// TIA Portal V15.1 export
// export: Created 2024-06-21T08:41:18.4574787Z, ExportSetting WithDefaults, DisplayName Totally Integrated Automation Portal, DisplayVersion V15.1 Update 5, DisplayName TIA Portal Openness, DisplayVersion V15.1 Update 5, DisplayName SINAMICS Startdrive Advanced, DisplayVersion V15.1, DisplayName G130, G150, S120, S150, SINAMICS MV, S210, DisplayVersion V15.1, DisplayName G110M, G120, G120C, G120D, G120P, DisplayVersion V15.1, DisplayName STEP 7 Professional, DisplayVersion V15.1 Update 5, DisplayName STEP 7 Safety, DisplayVersion V15.1, DisplayName WinCC Professional, DisplayVersion V15.1 Update 5, DisplayName SIMATIC Visualization Architect, DisplayVersion V15.1
FUNCTION_BLOCK "LGBLiftTable2Pos1S3Det-C"   // FB6675, FBD
TITLE = LMovUnit2Pos2Det2W2S-G120CU240PN / LMovUnit2Pos2W2S-G120CU240PN / LGBLiftTable2Pos1S3Det-C
{ S7_Optimized_Access := 'TRUE' }
AUTHOR : VCC
FAMILY : Tooling
VERSION : 0.0.0.0
// =============================================================================
// This module will be used for a unit with 2 stop positions, 2 speeds and controlled by a
// Siemens G120 PN frequency converter.
// It will get commands from higher level, evaluate the status of the interlock
// and give a finished in return when the task is completed.
// It will get commands from higher level, evaluate the status of the interlock
// and give a finished in return when the task is completed.
// ============================================================================
// stored: AutoNumber false, IsIECCheckEnabled false, IsRetainMemResEnabled false, MemoryReserve 100, SetENOAutomatically False, UDAEnableTagReadback false
   VAR_INPUT
      I_PosSet { ExternalAccessible := 'False'; ExternalVisible := 'False'; ExternalWritable := 'False'} : Bool;   // Position Set detection or summary / Position Set Detection / Position Set Detection 1
      I_PosSetCheck { ExternalAccessible := 'False'; ExternalVisible := 'False'; ExternalWritable := 'False'} : Bool;   // Low Speed Set / Low Speed Detection Set / Position Set Detection 2
      I_PosRes { ExternalAccessible := 'False'; ExternalVisible := 'False'; ExternalWritable := 'False'} : Bool;   // Position Reset detection or summary / Position Reset Detection / Position Reset Detection 1
      I_PosResCheck { ExternalAccessible := 'False'; ExternalVisible := 'False'; ExternalWritable := 'False'} : Bool;   // Low Speed Res / Low Speed Detection Reset / Position Reset Detection 2
      I_BrakeReleased { ExternalAccessible := 'False'; ExternalVisible := 'False'; ExternalWritable := 'False'} : Bool;   // Feedback from brake contactor
      I_SetBegin { ExternalAccessible := 'False'; ExternalVisible := 'False'; ExternalWritable := 'False'} : Bool;   // Function Set begin selection
      I_ResBegin { ExternalAccessible := 'False'; ExternalVisible := 'False'; ExternalWritable := 'False'} : Bool;   // Function Reset begin selection
      I_PBSet { ExternalAccessible := 'False'; ExternalVisible := 'False'; ExternalWritable := 'False'} : Bool;   // Push button for Set direction (used in manual with button OP panels ) / Push button for Set direction used in manual
      I_PBReset { ExternalAccessible := 'False'; ExternalVisible := 'False'; ExternalWritable := 'False'} : Bool;   // Push button for reset direcion (used in manual with pushbutton OP panels) / Push button for reset direcion used in manual
      I_SetIntlkOK { ExternalAccessible := 'False'; ExternalVisible := 'False'; ExternalWritable := 'False'} : Bool;   // Set Interlock
      I_ResIntlkOK { ExternalAccessible := 'False'; ExternalVisible := 'False'; ExternalWritable := 'False'} : Bool;   // Reset Interlock
      I_MotorProtection { ExternalAccessible := 'False'; ExternalVisible := 'False'; ExternalWritable := 'False'} : Bool;   // Motor protection
      I_SafetySwitch { ExternalAccessible := 'False'; ExternalVisible := 'False'; ExternalWritable := 'False'} : Bool;   // Safety switch
      I_SafetyOk { ExternalAccessible := 'False'; ExternalVisible := 'False'; ExternalWritable := 'False'} : Bool;   // Safety Ok
      I_MotionStopOk { ExternalAccessible := 'False'; ExternalVisible := 'False'; ExternalWritable := 'False'} : Bool;   // Safety Ok / The motion stop is Ok
   END_VAR
   VAR_OUTPUT
      O_SetContactor { ExternalAccessible := 'False'; ExternalVisible := 'False'; ExternalWritable := 'False'} : Bool;   // Activate set contactor
      O_ResetContactor { ExternalAccessible := 'False'; ExternalVisible := 'False'; ExternalWritable := 'False'} : Bool;   // Activate Reset contactor
      O_ReleaseBrakeContactor { ExternalAccessible := 'False'; ExternalVisible := 'False'; ExternalWritable := 'False'} : Bool;   // Release Brake
      O_Active { ExternalAccessible := 'False'; ExternalVisible := 'False'; ExternalWritable := 'False'} : Bool;   // Motor Loop Active / Motor Active
      O_SetPos { ExternalAccessible := 'False'; ExternalVisible := 'False'; ExternalWritable := 'False'} : Bool;   // Summary In Position Set / In Position Set
      O_ResPos { ExternalAccessible := 'False'; ExternalVisible := 'False'; ExternalWritable := 'False'} : Bool;   // Summary In Position Reset / In Position Reset
      O_FuncRunning { ExternalAccessible := 'False'; ExternalVisible := 'False'; ExternalWritable := 'False'} : Bool;   // Signal that the function is busy
      O_SetFinished { ExternalAccessible := 'False'; ExternalVisible := 'False'; ExternalWritable := 'False'} : Bool;   // Function Set finished to Master Sequencing
      O_ResFinished { ExternalAccessible := 'False'; ExternalVisible := 'False'; ExternalWritable := 'False'} : Bool;   // Function Reset finished to Master Sequencing
      O_LEDSet { ExternalAccessible := 'False'; ExternalVisible := 'False'; ExternalWritable := 'False'} : Bool;   // Ledindication / Led indication for Set
      O_LEDRes { ExternalAccessible := 'False'; ExternalVisible := 'False'; ExternalWritable := 'False'} : Bool;   // Ledindication / Led indication for Reset
      O_AlarmABCondition { ExternalAccessible := 'False'; ExternalVisible := 'False'; ExternalWritable := 'False'} : Bool;   // Alarm AB condition
      O_AlarmA { ExternalAccessible := 'False'; ExternalVisible := 'False'; ExternalWritable := 'False'} : Bool;   // Summation Alarm A of roller. / Alarm A
      O_AlarmB { ExternalAccessible := 'False'; ExternalVisible := 'False'; ExternalWritable := 'False'} : Bool;   // Summation Alarm B of roller. / Alarm B
      O_AlarmC { ExternalAccessible := 'False'; ExternalVisible := 'False'; ExternalWritable := 'False'} : Bool;   // Summation Alarm C of roller. / Alarm C
      O_AlarmD { ExternalAccessible := 'False'; ExternalVisible := 'False'; ExternalWritable := 'False'} : Bool;   // Summation Alarm D of roller. / Alarm D
      H_AlarmDWord { ExternalAccessible := 'False'; ExternalVisible := 'False'; ExternalWritable := 'False'} : DWord;   // HMI Animation of the alarms of the roller / Alarm Word
   END_VAR
   VAR_IN_OUT
      IO_Modes : "Modes";   // Modes
      C_Config : "LiftTable2Pos1S3Det-C-Config";   // Config
      H_HMI : "H_HMI";   // Animation
      "H_GBLiftTable2Pos1S3Det-C" : "H_GBLiftTable2Pos1S3Det-C";   // Animation
   END_VAR
   VAR
      _MovFunc2Pos { ExternalAccessible := 'False'; ExternalVisible := 'False'; ExternalWritable := 'False'} : "LMovFnc2Pos";   // Move function 2 positioner / FB
      _StopPos { ExternalAccessible := 'False'; ExternalVisible := 'False'; ExternalWritable := 'False'} : "L2StopPos";   // FB
      _Motor { ExternalAccessible := 'False'; ExternalVisible := 'False'; ExternalWritable := 'False'} : "LGBMotor2W1S-C";   // FB
      _SetDetMissing { ExternalAccessible := 'False'; ExternalVisible := 'False'; ExternalWritable := 'False'} : "LTimer";   // Timer
      _ResDetMissing { ExternalAccessible := 'False'; ExternalVisible := 'False'; ExternalWritable := 'False'} : "LTimer";   // Timer
      H_FncSelInHMI { ExternalAccessible := 'False'; ExternalVisible := 'False'; ExternalWritable := 'False'} : Bool;
      AA_MotorProtection { ExternalAccessible := 'False'; ExternalVisible := 'False'; ExternalWritable := 'False'} : Bool;   // Motor protection alarm / Motorprotection Not Ok / Motor Protection Tripped / Motorskyddsbrytare Ej Ok
      AA_SafetySwitch { ExternalAccessible := 'False'; ExternalVisible := 'False'; ExternalWritable := 'False'} : Bool;   // Safety Switch alarm / Safety Switch Not Ok / Säkerhetsbrytare Ej Ok
      AB_BrakeFbk { ExternalAccessible := 'False'; ExternalVisible := 'False'; ExternalWritable := 'False'} : Bool;   // Safety Switch Not Ok / Brake feedback Nok / Säkerhetsbrytare Ej Ok
      AB_KeepPosSetAlm { ExternalAccessible := 'False'; ExternalVisible := 'False'; ExternalWritable := 'False'} : Bool;   // 0000: Keep position set alarm / Position Supervision Set Position / Lost Set Position / Positionsövervakning Set Läge
      AB_KeepPosResAlm { ExternalAccessible := 'False'; ExternalVisible := 'False'; ExternalWritable := 'False'} : Bool;   // 0000: Keep position reset alarm / Position Supervision Reset Position / Lost Reset Position / Positionsövervakning Reset Läge
      AB_OvtSetAlm { ExternalAccessible := 'False'; ExternalVisible := 'False'; ExternalWritable := 'False'} : Bool;   // 0000: Overtime set alarm / Timeout Set / TimeOut Set Direction / Tidsövervakning Set
      AB_OvtResAlm { ExternalAccessible := 'False'; ExternalVisible := 'False'; ExternalWritable := 'False'} : Bool;   // 0000: Overtime reset alarm / Timeout Reset / TimeOut Reset Direction / Tidsövervakning Reset
      AB_TwoDetAlm { ExternalAccessible := 'False'; ExternalVisible := 'False'; ExternalWritable := 'False'} : Bool;   // 0000: Two detection alarm / Set Reset Activated Simultaneously / Detection Set & Reset Activated Simultaneously / Set Reset Påverkade Samtidigt
      AB_SetDet1Missing { ExternalAccessible := 'False'; ExternalVisible := 'False'; ExternalWritable := 'False'} : Bool;   // 0000: Two detection alarm / Set Detector 1 Signal Missing / Set Detector Signal Missing / Setgivare 1 signal saknas
      AB_SetDet2Missing { ExternalAccessible := 'False'; ExternalVisible := 'False'; ExternalWritable := 'False'} : Bool;   // 0000: Two detection alarm / Set Detector 2 Signal Missing / Set Check Detector Signal Missing / Setgivare 2 signal saknas
      AB_ResDet1Missing { ExternalAccessible := 'False'; ExternalVisible := 'False'; ExternalWritable := 'False'} : Bool;   // 0000: Two detection alarm / Resetgivare 1 signal saknas / Reset Detector Signal Missing
      AB_ResDet2Missing { ExternalAccessible := 'False'; ExternalVisible := 'False'; ExternalWritable := 'False'} : Bool;   // 0000: Two detection alarm / Resetgivare 2 signal saknas / Reset Check Detector Signal Missing
      AC_KeepPosSetAlm { ExternalAccessible := 'False'; ExternalVisible := 'False'; ExternalWritable := 'False'} : Bool;   // 0000: Keep position set alarm / Lost Set Position / Tappat Set Position
      AC_KeepPosResAlm { ExternalAccessible := 'False'; ExternalVisible := 'False'; ExternalWritable := 'False'} : Bool;   // 0000: Keep position reset alarm / Lost Reset Position / Tappat Reset Position
      AC_OvtSetAlm { ExternalAccessible := 'False'; ExternalVisible := 'False'; ExternalWritable := 'False'} : Bool;   // 0000: Overtime set alarm / Timeout Set / TimeOut Set Direction / Tidsövervakning Set
      AC_OvtResAlm { ExternalAccessible := 'False'; ExternalVisible := 'False'; ExternalWritable := 'False'} : Bool;   // 0000: Overtime reset alarm / Timeout Reset / TimeOut Reset Direction / Tidsövervakning Reset
      AC_TwoDetAlm { ExternalAccessible := 'False'; ExternalVisible := 'False'; ExternalWritable := 'False'} : Bool;   // 0000: Two detection alarm / Set Reset Activated Simultaneously / Detection Set & Reset Activated Simultaneously / Set Reset Påverkade Samtidigt
      AC_SetDet1Missing { ExternalAccessible := 'False'; ExternalVisible := 'False'; ExternalWritable := 'False'} : Bool;   // 0000: Two detection alarm / Set Detector 1 Signal Missing / Set Detector Signal Missing / Setgivare 1 signal saknas
      AC_SetDet2Missing { ExternalAccessible := 'False'; ExternalVisible := 'False'; ExternalWritable := 'False'} : Bool;   // 0000: Two detection alarm / Set Detector 2 Signal Missing / Set Check Detector Signal Missing / Setgivare 2 signal saknas
      AC_ResDet1Missing { ExternalAccessible := 'False'; ExternalVisible := 'False'; ExternalWritable := 'False'} : Bool;   // 0000: Two detection alarm / Resetgivare 1 signal saknas / Reset Detector Signal Missing
      AC_ResDet2Missing { ExternalAccessible := 'False'; ExternalVisible := 'False'; ExternalWritable := 'False'} : Bool;   // 0000: Two detection alarm / Resetgivare 2 signal saknas / Reset Check Detector Signal Missing
      AD_OvtSetWarn { ExternalAccessible := 'False'; ExternalVisible := 'False'; ExternalWritable := 'False'} : Bool;   // 0000: Overtime set warning / Timeout Set / TimeOut Set Direction / Tidsövervakning Set
      AD_OvtResWarn { ExternalAccessible := 'False'; ExternalVisible := 'False'; ExternalWritable := 'False'} : Bool;   // 0000: Overtime reset warning / Timeout Reset / TimeOut Reset Direction / Tidsövervakning Reset
      AD_IntlkSetAlm { ExternalAccessible := 'False'; ExternalVisible := 'False'; ExternalWritable := 'False'} : Bool;   // 0000: Interlock Set alarm / Interlock Set
      AD_IntlkResAlm { ExternalAccessible := 'False'; ExternalVisible := 'False'; ExternalWritable := 'False'} : Bool;   // 0000: Interlock Reset alarm / Interlock Reset
      AD_MotionStop { ExternalAccessible := 'False'; ExternalVisible := 'False'; ExternalWritable := 'False'} : Bool;   // Motion Stop
      AC_ConfigCalibrationAlm { ExternalAccessible := 'False'; ExternalVisible := 'False'; ExternalWritable := 'False'} : Bool;   // The Config values for Warming/Alarm time must be ALL zero or ALL different from zero
      AD_CalibrationWarn { ExternalAccessible := 'False'; ExternalVisible := 'False'; ExternalWritable := 'False'} : Bool;   // No High speed selected so Calibration is not possible
      SafetyOk { ExternalAccessible := 'False'; ExternalVisible := 'False'; ExternalWritable := 'False'} : Bool;   // Safety Ok
      SetPos { ExternalAccessible := 'False'; ExternalVisible := 'False'; ExternalWritable := 'False'} : Bool;   // Set position
      ResPos { ExternalAccessible := 'False'; ExternalVisible := 'False'; ExternalWritable := 'False'} : Bool;   // Reset position
      AlarmA { ExternalAccessible := 'False'; ExternalVisible := 'False'; ExternalWritable := 'False'} : Bool;   // Summation Alarm A / Alarm A
      AlarmB { ExternalAccessible := 'False'; ExternalVisible := 'False'; ExternalWritable := 'False'} : Bool;   // Summation Alarm B / Alarm B
      AlarmC { ExternalAccessible := 'False'; ExternalVisible := 'False'; ExternalWritable := 'False'} : Bool;   // Summation Alarm C / Alarm C
      AlarmD { ExternalAccessible := 'False'; ExternalVisible := 'False'; ExternalWritable := 'False'} : Bool;   // Summation Alarm D / Alarm D
      SetIntlkOK { ExternalAccessible := 'False'; ExternalVisible := 'False'; ExternalWritable := 'False'} : Bool;   // Set Interlock
      ResIntlkOK { ExternalAccessible := 'False'; ExternalVisible := 'False'; ExternalWritable := 'False'} : Bool;   // Reset Interlock
      FuncRunning { ExternalAccessible := 'False'; ExternalVisible := 'False'; ExternalWritable := 'False'} : Bool;   // Function running
      MovFuncAlmCond { ExternalAccessible := 'False'; ExternalVisible := 'False'; ExternalWritable := 'False'} : Bool;   // Move function alarm condition / Move function Alarm Condition
      StopPosAlmCond { ExternalAccessible := 'False'; ExternalVisible := 'False'; ExternalWritable := 'False'} : Bool;   // Stop posistion alarm condition / Stop posistion Alarm Condition
      KeepPosSetAlm { ExternalAccessible := 'False'; ExternalVisible := 'False'; ExternalWritable := 'False'} : Bool;   // Keep position set alarm / Alarm Keep Position Set Position / Larm Positions Övervakning Set Läge
      KeepPosResAlm { ExternalAccessible := 'False'; ExternalVisible := 'False'; ExternalWritable := 'False'} : Bool;   // Keep position reset alarm / Position Supervision Reset Position / Positions Övervakning Reset Läge
      OvtSetAlm { ExternalAccessible := 'False'; ExternalVisible := 'False'; ExternalWritable := 'False'} : Bool;   // Overtime set alarm / Timeout Set / Tidsövervakning Set
      OvtResAlm { ExternalAccessible := 'False'; ExternalVisible := 'False'; ExternalWritable := 'False'} : Bool;   // Overtime reset alarm / Overtime reset Alarm
      TwoDetAlm { ExternalAccessible := 'False'; ExternalVisible := 'False'; ExternalWritable := 'False'} : Bool;   // Two detection alarm / Set Reset Activated Simultaneously / Set Reset Påverkade Samtidigt
      OneSetDetMissing { ExternalAccessible := 'False'; ExternalVisible := 'False'; ExternalWritable := 'False'} : Bool;   // Two detection alarm / One Set detector is missing
      OneResDetMissing { ExternalAccessible := 'False'; ExternalVisible := 'False'; ExternalWritable := 'False'} : Bool;   // Two detection alarm / One Reset detector is missing
      DetectorMissing { ExternalAccessible := 'False'; ExternalVisible := 'False'; ExternalWritable := 'False'} : Bool;   // Two detection alarm / One detector is missing
      MotorLoopAlarmCond { ExternalAccessible := 'False'; ExternalVisible := 'False'; ExternalWritable := 'False'} : Bool;   // Motor loop alarm condition / Motor loop Alarm Condition
      MotorLoopActive { ExternalAccessible := 'False'; ExternalVisible := 'False'; ExternalWritable := 'False'} : Bool;   // Motor Loop Active
      AlarmABCondition { ExternalAccessible := 'False'; ExternalVisible := 'False'; ExternalWritable := 'False'} : Bool;   // Alarm AB Condition
      MotorCmdSet { ExternalAccessible := 'False'; ExternalVisible := 'False'; ExternalWritable := 'False'} : Bool;   // Command high speed to motorloop set / Command to motorloop set
      MotorCmdRes { ExternalAccessible := 'False'; ExternalVisible := 'False'; ExternalWritable := 'False'} : Bool;   // Command high speed to motorloop reset / Command to motorloop reset
      SetContactor { ExternalAccessible := 'False'; ExternalVisible := 'False'; ExternalWritable := 'False'} : Bool;   // Activate set contactor
      ResetContactor { ExternalAccessible := 'False'; ExternalVisible := 'False'; ExternalWritable := 'False'} : Bool;   // Activate Reset contactor
      ReleaseBrakeContactor { ExternalAccessible := 'False'; ExternalVisible := 'False'; ExternalWritable := 'False'} : Bool;   // Activate Reset contactor / Release Brake contactor
      SetPosDelayd { ExternalAccessible := 'False'; ExternalVisible := 'False'; ExternalWritable := 'False'} : Bool;   // Set Position Delayed
      ResPosDelayd { ExternalAccessible := 'False'; ExternalVisible := 'False'; ExternalWritable := 'False'} : Bool;   // Reset Position Delayed
      PosSetDelayTimer { ExternalAccessible := 'False'; ExternalVisible := 'False'; ExternalWritable := 'False'} : "LTimer";   // FB
      PosResDelayTimer { ExternalAccessible := 'False'; ExternalVisible := 'False'; ExternalWritable := 'False'} : "LTimer";   // FB
   END_VAR
   VAR_TEMP
      H_HMITemp : "H_HMI";   // Animation
      H_HMIMotor : "H_HMI";   // Temp
   END_VAR
   VAR_TEMP   // added for the SCL form of the ladder/FBD networks
      _w1 : Bool;
   END_VAR
BEGIN

REGION Network 1: **** 1 - Inputs **** Set Position Delay Timer
   // Set Position Delay Timer
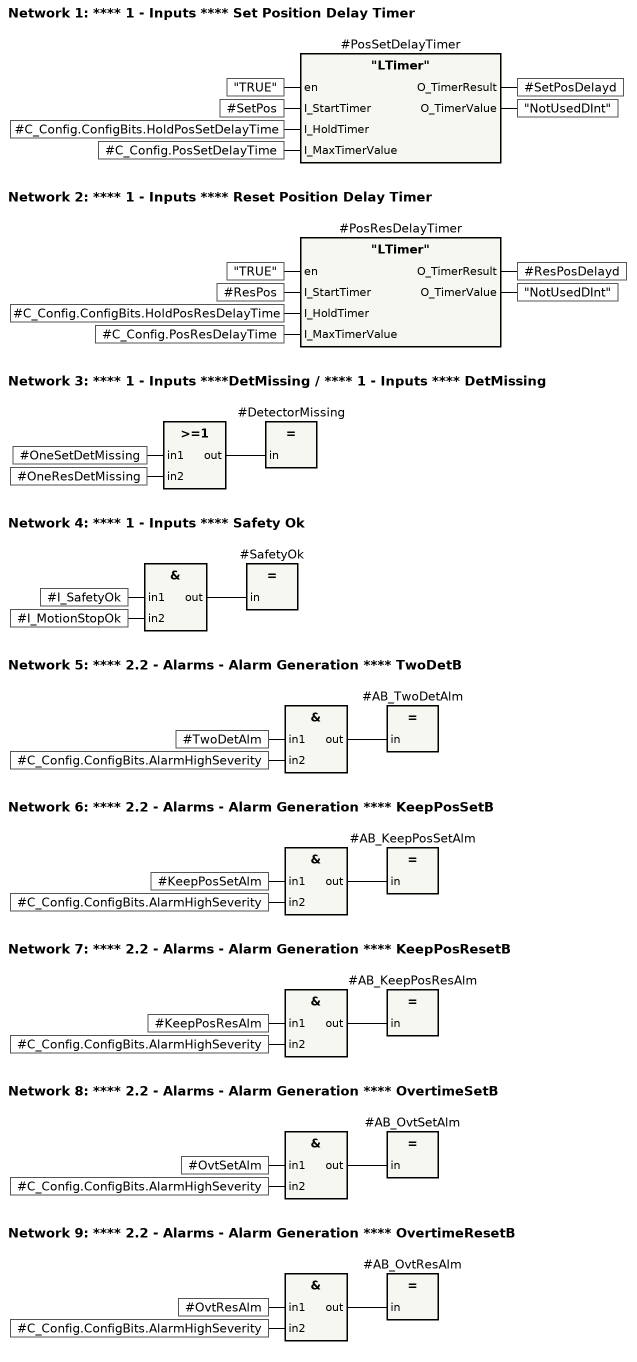
   IF "TRUE" THEN
       #PosSetDelayTimer(I_StartTimer := #SetPos,   // "LTimer"
                         I_HoldTimer := #C_Config.ConfigBits.HoldPosSetDelayTime,
                         I_MaxTimerValue := #C_Config.PosSetDelayTime,
                         O_TimerResult => #SetPosDelayd,
                         O_TimerValue => "NotUsedDInt");
   END_IF;
END_REGION

REGION Network 2: **** 1 - Inputs **** Reset Position Delay Timer
   // Reset Position Delay Timer
   IF "TRUE" THEN
       #PosResDelayTimer(I_StartTimer := #ResPos,   // "LTimer"
                         I_HoldTimer := #C_Config.ConfigBits.HoldPosResDelayTime,
                         I_MaxTimerValue := #C_Config.PosResDelayTime,
                         O_TimerResult => #ResPosDelayd,
                         O_TimerValue => "NotUsedDInt");
   END_IF;
END_REGION

REGION Network 3: **** 1 - Inputs ****DetMissing / **** 1 - Inputs **** DetMissing
   // Disable other Alarms when a detector is missing
   #DetectorMissing := #OneSetDetMissing OR #OneResDetMissing;
END_REGION

REGION Network 4: **** 1 - Inputs **** Safety Ok
   #SafetyOk := #I_SafetyOk AND #I_MotionStopOk;
END_REGION

REGION Network 5: **** 2.2 - Alarms - Alarm Generation **** TwoDetB
   // Two Detection B Alarm
   #AB_TwoDetAlm := #TwoDetAlm AND #C_Config.ConfigBits.AlarmHighSeverity;
END_REGION

REGION Network 6: **** 2.2 - Alarms - Alarm Generation **** KeepPosSetB
   // Keep position Set B Alarm
   #AB_KeepPosSetAlm := #KeepPosSetAlm AND #C_Config.ConfigBits.AlarmHighSeverity;
END_REGION

REGION Network 7: **** 2.2 - Alarms - Alarm Generation **** KeepPosResetB
   // Keep position reset B Alarm
   #AB_KeepPosResAlm := #KeepPosResAlm AND #C_Config.ConfigBits.AlarmHighSeverity;
END_REGION

REGION Network 8: **** 2.2 - Alarms - Alarm Generation **** OvertimeSetB
   // Overtime set B Alarm
   #AB_OvtSetAlm := #OvtSetAlm AND #C_Config.ConfigBits.AlarmHighSeverity;
END_REGION

REGION Network 9: **** 2.2 - Alarms - Alarm Generation **** OvertimeResetB
   // Overtime reset B Alarm
   #AB_OvtResAlm := #OvtResAlm AND #C_Config.ConfigBits.AlarmHighSeverity;
END_REGION

REGION Network 10: **** 2.2 - Alarms - Alarm Generation ****SetDetMissing
   // Any Set detector missing
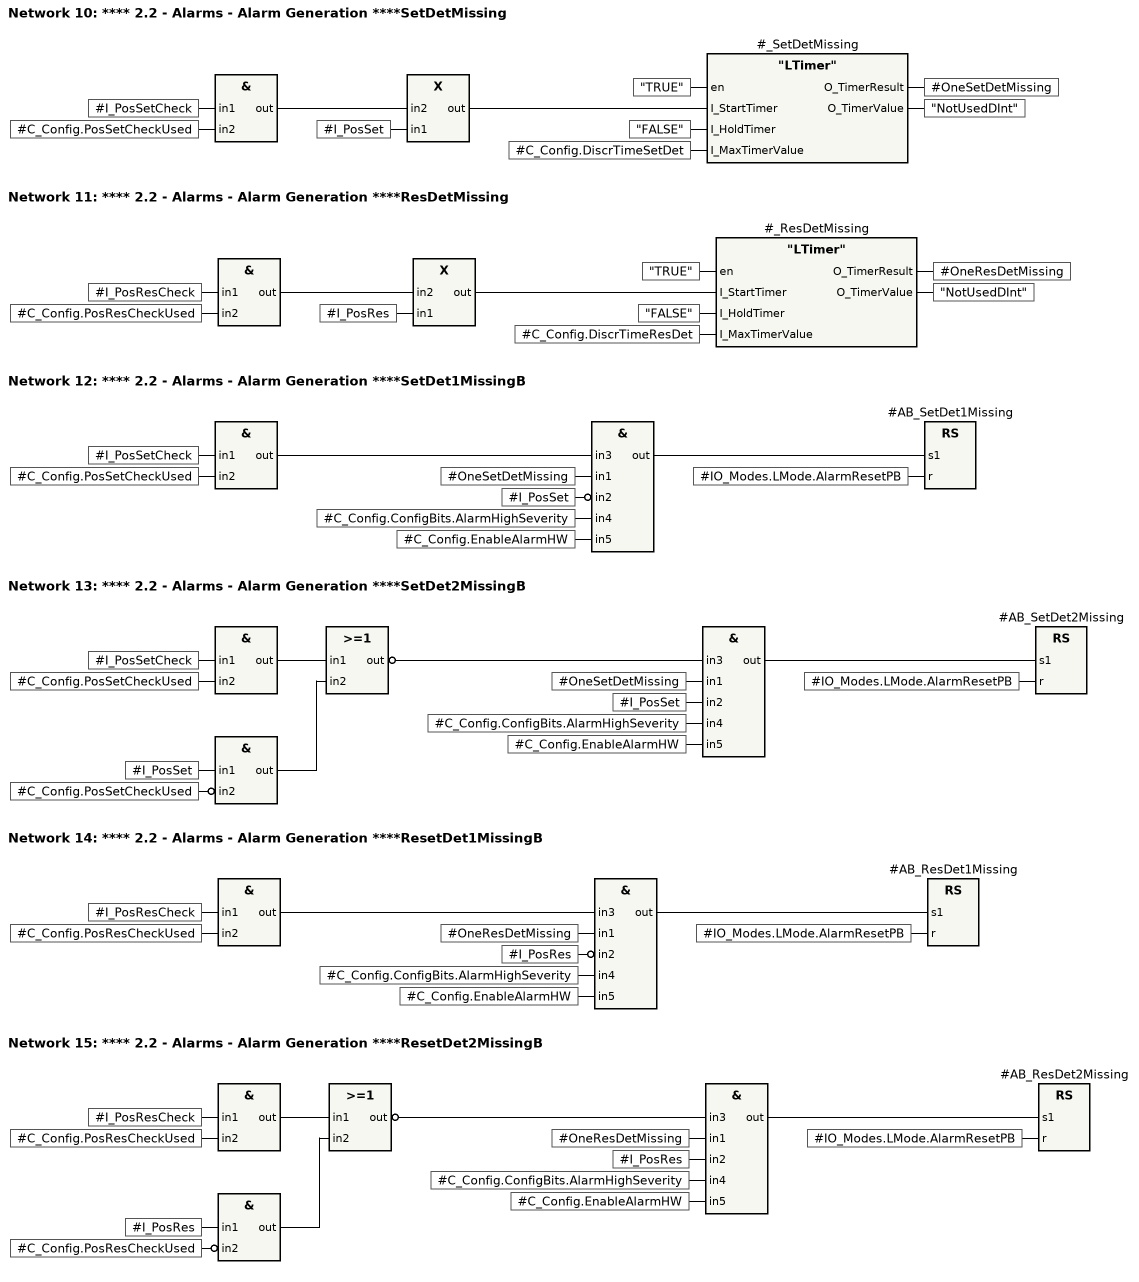
   IF "TRUE" THEN
       #_SetDetMissing(I_StartTimer := (#I_PosSetCheck AND #C_Config.PosSetCheckUsed) XOR #I_PosSet,   // "LTimer"
                       I_HoldTimer := "FALSE",
                       I_MaxTimerValue := #C_Config.DiscrTimeSetDet,
                       O_TimerResult => #OneSetDetMissing,
                       O_TimerValue => "NotUsedDInt");
   END_IF;
END_REGION

REGION Network 11: **** 2.2 - Alarms - Alarm Generation ****ResDetMissing
   // Any Reset detector missing
   IF "TRUE" THEN
       #_ResDetMissing(I_StartTimer := (#I_PosResCheck AND #C_Config.PosResCheckUsed) XOR #I_PosRes,   // "LTimer"
                       I_HoldTimer := "FALSE",
                       I_MaxTimerValue := #C_Config.DiscrTimeResDet,
                       O_TimerResult => #OneResDetMissing,
                       O_TimerValue => "NotUsedDInt");
   END_IF;
END_REGION

REGION Network 12: **** 2.2 - Alarms - Alarm Generation ****SetDet1MissingB
   // Set detector 1 missing
   IF #IO_Modes.LMode.AlarmResetPB THEN
       #AB_SetDet1Missing := FALSE;   // RS flip-flop
   END_IF;
   IF #I_PosSetCheck AND #C_Config.PosSetCheckUsed AND #OneSetDetMissing AND NOT #I_PosSet AND #C_Config.ConfigBits.AlarmHighSeverity AND #C_Config.EnableAlarmHW THEN
       #AB_SetDet1Missing := TRUE;
   END_IF;
END_REGION

REGION Network 13: **** 2.2 - Alarms - Alarm Generation ****SetDet2MissingB
   // Set detector 2 missing
   IF #IO_Modes.LMode.AlarmResetPB THEN
       #AB_SetDet2Missing := FALSE;   // RS flip-flop
   END_IF;
   IF NOT ((#I_PosSetCheck AND #C_Config.PosSetCheckUsed) OR (#I_PosSet AND NOT #C_Config.PosSetCheckUsed)) AND #OneSetDetMissing AND #I_PosSet AND #C_Config.ConfigBits.AlarmHighSeverity AND #C_Config.EnableAlarmHW THEN
       #AB_SetDet2Missing := TRUE;
   END_IF;
END_REGION

REGION Network 14: **** 2.2 - Alarms - Alarm Generation ****ResetDet1MissingB
   // Reset detector 1 missing
   IF #IO_Modes.LMode.AlarmResetPB THEN
       #AB_ResDet1Missing := FALSE;   // RS flip-flop
   END_IF;
   IF #I_PosResCheck AND #C_Config.PosResCheckUsed AND #OneResDetMissing AND NOT #I_PosRes AND #C_Config.ConfigBits.AlarmHighSeverity AND #C_Config.EnableAlarmHW THEN
       #AB_ResDet1Missing := TRUE;
   END_IF;
END_REGION

REGION Network 15: **** 2.2 - Alarms - Alarm Generation ****ResetDet2MissingB
   // Reset detector 2 missing
   IF #IO_Modes.LMode.AlarmResetPB THEN
       #AB_ResDet2Missing := FALSE;   // RS flip-flop
   END_IF;
   IF NOT ((#I_PosResCheck AND #C_Config.PosResCheckUsed) OR (#I_PosRes AND NOT #C_Config.PosResCheckUsed)) AND #OneResDetMissing AND #I_PosRes AND #C_Config.ConfigBits.AlarmHighSeverity AND #C_Config.EnableAlarmHW THEN
       #AB_ResDet2Missing := TRUE;
   END_IF;
END_REGION

REGION Network 16: **** 2.2 - Alarms - Alarm Generation **** TwoDetC
   // Two Detection C Alarm
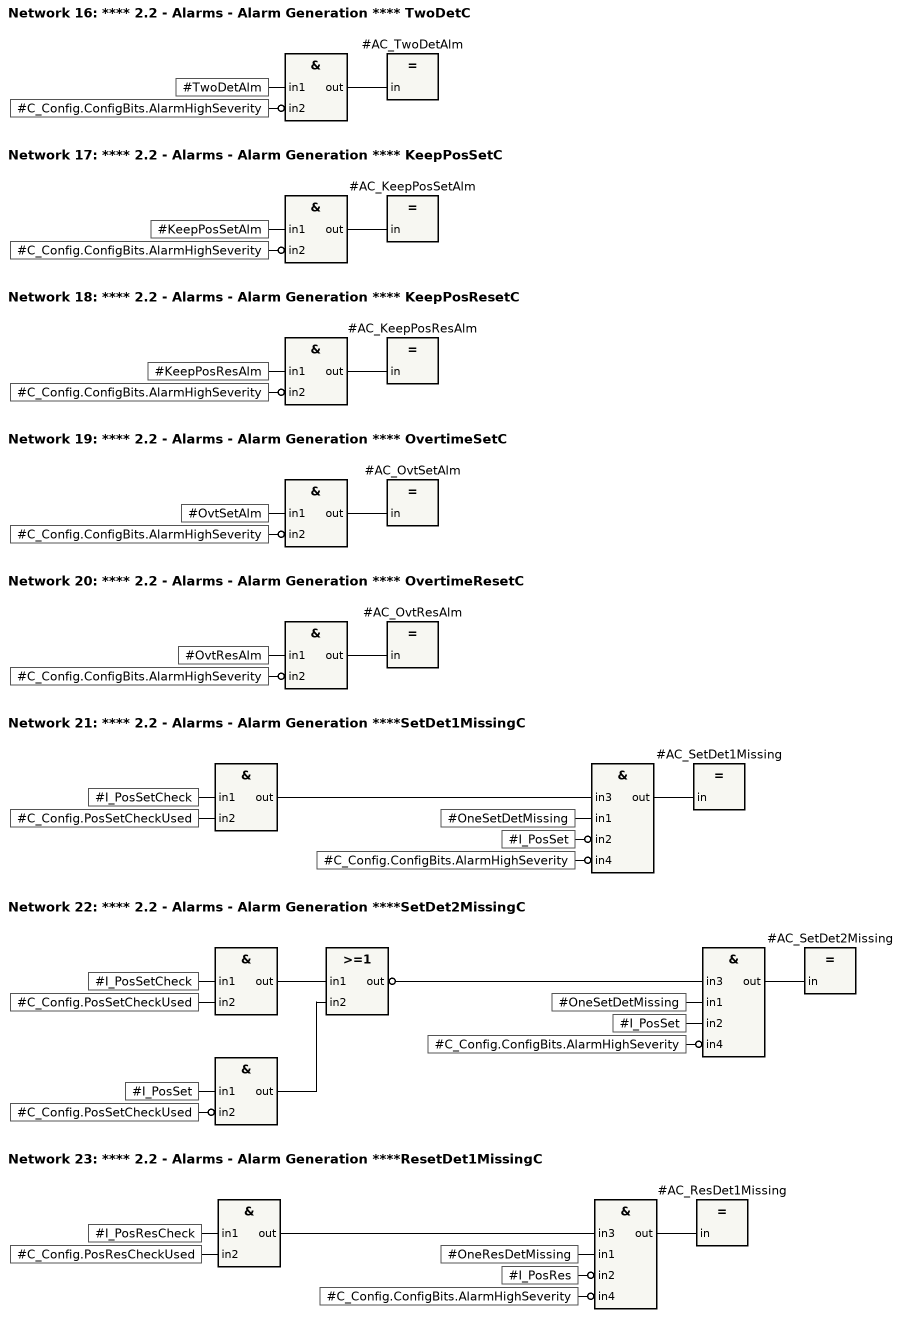
   #AC_TwoDetAlm := #TwoDetAlm AND NOT #C_Config.ConfigBits.AlarmHighSeverity;
END_REGION

REGION Network 17: **** 2.2 - Alarms - Alarm Generation **** KeepPosSetC
   // Keep position Set C Alarm
   #AC_KeepPosSetAlm := #KeepPosSetAlm AND NOT #C_Config.ConfigBits.AlarmHighSeverity;
END_REGION

REGION Network 18: **** 2.2 - Alarms - Alarm Generation **** KeepPosResetC
   // Keep position reset C Alarm
   #AC_KeepPosResAlm := #KeepPosResAlm AND NOT #C_Config.ConfigBits.AlarmHighSeverity;
END_REGION

REGION Network 19: **** 2.2 - Alarms - Alarm Generation **** OvertimeSetC
   // Overtime set C Alarm
   #AC_OvtSetAlm := #OvtSetAlm AND NOT #C_Config.ConfigBits.AlarmHighSeverity;
END_REGION

REGION Network 20: **** 2.2 - Alarms - Alarm Generation **** OvertimeResetC
   // Overtime reset C Alarm
   #AC_OvtResAlm := #OvtResAlm AND NOT #C_Config.ConfigBits.AlarmHighSeverity;
END_REGION

REGION Network 21: **** 2.2 - Alarms - Alarm Generation ****SetDet1MissingC
   // Set detector 1 missing
   #AC_SetDet1Missing := #I_PosSetCheck AND #C_Config.PosSetCheckUsed AND #OneSetDetMissing AND NOT #I_PosSet AND NOT #C_Config.ConfigBits.AlarmHighSeverity;
END_REGION

REGION Network 22: **** 2.2 - Alarms - Alarm Generation ****SetDet2MissingC
   // Set detector 2 missing
   #AC_SetDet2Missing := NOT ((#I_PosSetCheck AND #C_Config.PosSetCheckUsed) OR (#I_PosSet AND NOT #C_Config.PosSetCheckUsed)) AND #OneSetDetMissing AND #I_PosSet AND NOT #C_Config.ConfigBits.AlarmHighSeverity;
END_REGION

REGION Network 23: **** 2.2 - Alarms - Alarm Generation ****ResetDet1MissingC
   // Reset detector 1 missing
   #AC_ResDet1Missing := #I_PosResCheck AND #C_Config.PosResCheckUsed AND #OneResDetMissing AND NOT #I_PosRes AND NOT #C_Config.ConfigBits.AlarmHighSeverity;
END_REGION

REGION Network 24: **** 2.2 - Alarms - Alarm Generation ****ResetDet2MissingC
   // Reset detector 2 missing
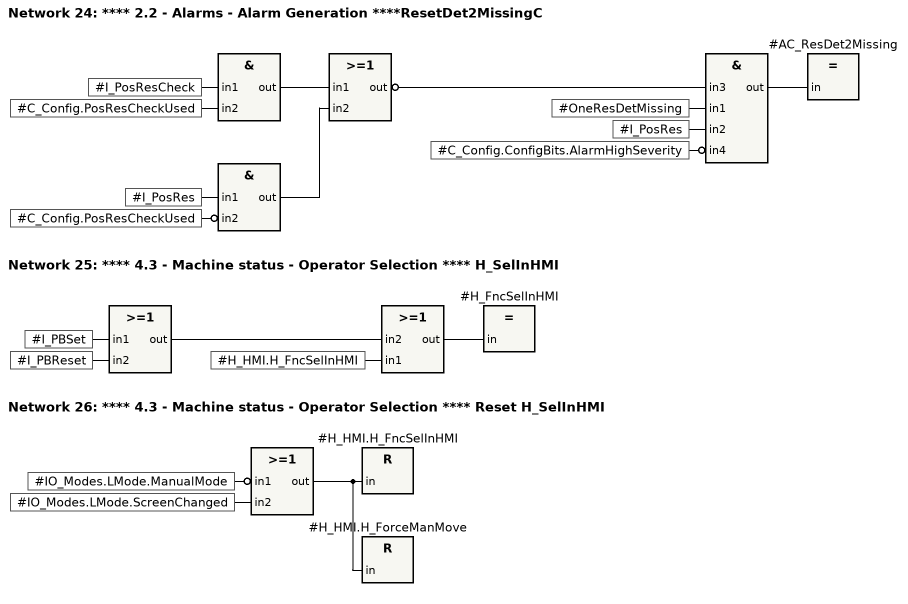
   #AC_ResDet2Missing := NOT ((#I_PosResCheck AND #C_Config.PosResCheckUsed) OR (#I_PosRes AND NOT #C_Config.PosResCheckUsed)) AND #OneResDetMissing AND #I_PosRes AND NOT #C_Config.ConfigBits.AlarmHighSeverity;
END_REGION

REGION Network 25: **** 4.3 - Machine status - Operator Selection **** H_SelInHMI
   #H_FncSelInHMI := #I_PBSet OR #I_PBReset OR #H_HMI.H_FncSelInHMI;
END_REGION

REGION Network 26: **** 4.3 - Machine status - Operator Selection **** Reset H_SelInHMI
   // Reset H_SelInHMI
   IF NOT #IO_Modes.LMode.ManualMode OR #IO_Modes.LMode.ScreenChanged THEN
       #H_HMI.H_FncSelInHMI := FALSE;
       #H_HMI.H_ForceManMove := FALSE;
   END_IF;
END_REGION

REGION Network 27: **** 4.6 - Machine status - Indication **** Icon Animation
   // Icon animation
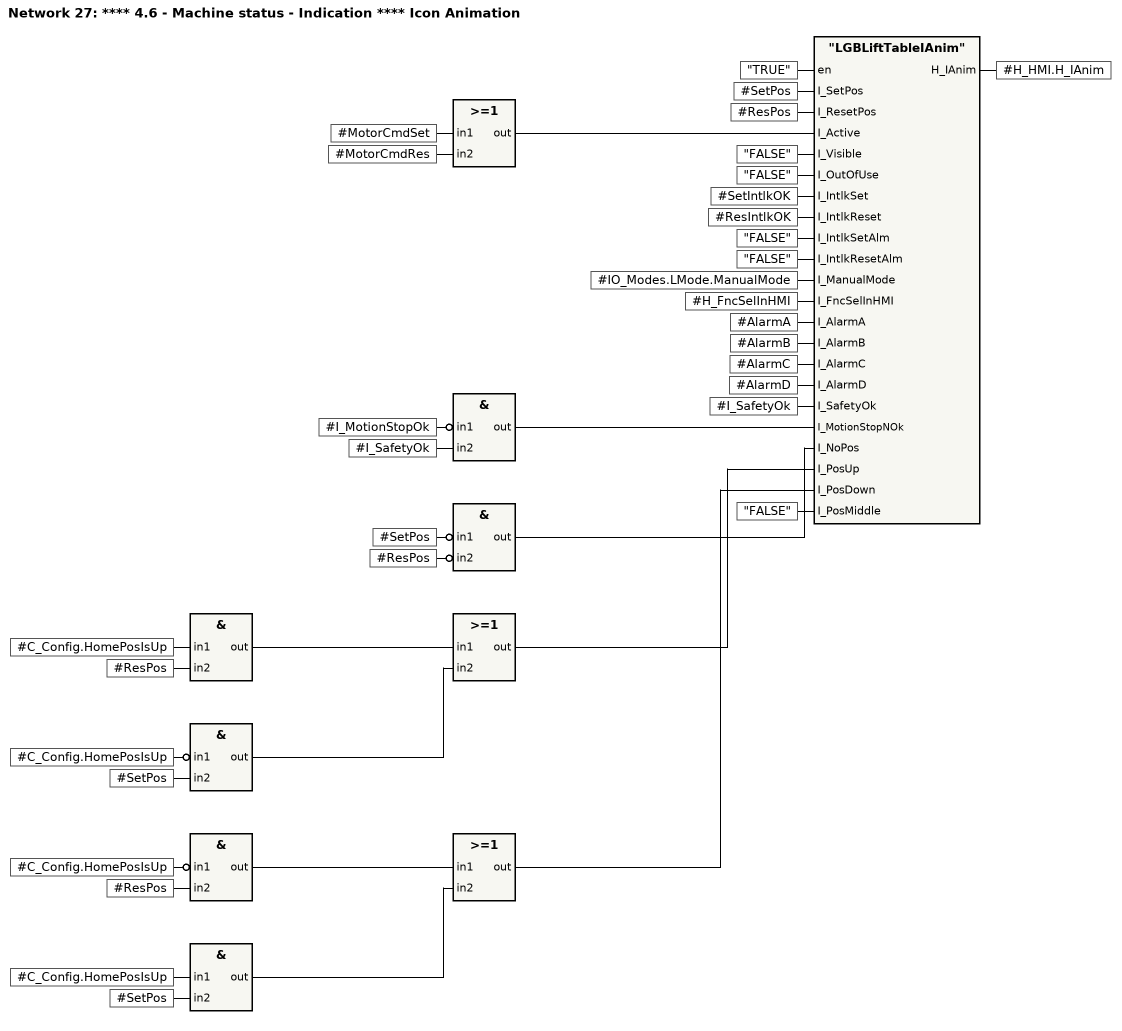
   IF "TRUE" THEN
       "LGBLiftTableIAnim"(I_SetPos := #SetPos,
                           I_ResetPos := #ResPos,
                           I_Active := #MotorCmdSet OR #MotorCmdRes,
                           I_Visible := "FALSE",
                           I_OutOfUse := "FALSE",
                           I_IntlkSet := #SetIntlkOK,
                           I_IntlkReset := #ResIntlkOK,
                           I_IntlkSetAlm := "FALSE",
                           I_IntlkResetAlm := "FALSE",
                           I_ManualMode := #IO_Modes.LMode.ManualMode,
                           I_FncSelInHMI := #H_FncSelInHMI,
                           I_AlarmA := #AlarmA,
                           I_AlarmB := #AlarmB,
                           I_AlarmC := #AlarmC,
                           I_AlarmD := #AlarmD,
                           I_SafetyOk := #I_SafetyOk,
                           I_MotionStopNOk := NOT #I_MotionStopOk AND #I_SafetyOk,
                           I_NoPos := NOT #SetPos AND NOT #ResPos,
                           I_PosUp := (#C_Config.HomePosIsUp AND #ResPos) OR (NOT #C_Config.HomePosIsUp AND #SetPos),
                           I_PosDown := (NOT #C_Config.HomePosIsUp AND #ResPos) OR (#C_Config.HomePosIsUp AND #SetPos),
                           I_PosMiddle := "FALSE",
                           H_IAnim => #H_HMI.H_IAnim);
   END_IF;
END_REGION

REGION Network 28: **** 4.6 - Machine status - Indication **** SetDet1IAnim / **** 4.6 - Machine status - Indication **** SetDetIAnim / **** 4.6 - Machine status - Indication **** DetSetIAnim
   // Icon animation
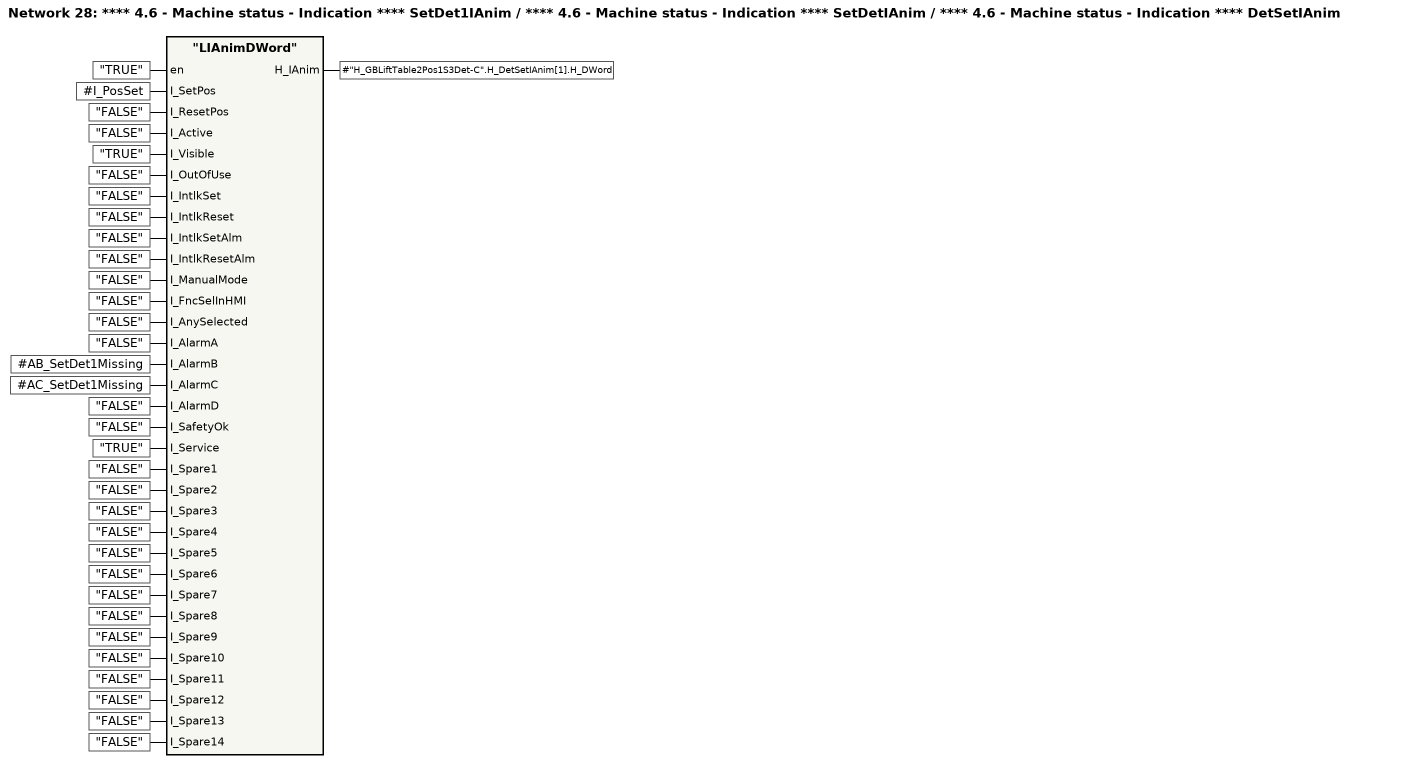
   IF "TRUE" THEN
       "LIAnimDWord"(I_SetPos := #I_PosSet,
                     I_ResetPos := "FALSE",
                     I_Active := "FALSE",
                     I_Visible := "TRUE",
                     I_OutOfUse := "FALSE",
                     I_IntlkSet := "FALSE",
                     I_IntlkReset := "FALSE",
                     I_IntlkSetAlm := "FALSE",
                     I_IntlkResetAlm := "FALSE",
                     I_ManualMode := "FALSE",
                     I_FncSelInHMI := "FALSE",
                     I_AnySelected := "FALSE",
                     I_AlarmA := "FALSE",
                     I_AlarmB := #AB_SetDet1Missing,
                     I_AlarmC := #AC_SetDet1Missing,
                     I_AlarmD := "FALSE",
                     I_SafetyOk := "FALSE",
                     I_Service := "TRUE",
                     I_Spare1 := "FALSE",
                     I_Spare2 := "FALSE",
                     I_Spare3 := "FALSE",
                     I_Spare4 := "FALSE",
                     I_Spare5 := "FALSE",
                     I_Spare6 := "FALSE",
                     I_Spare7 := "FALSE",
                     I_Spare8 := "FALSE",
                     I_Spare9 := "FALSE",
                     I_Spare10 := "FALSE",
                     I_Spare11 := "FALSE",
                     I_Spare12 := "FALSE",
                     I_Spare13 := "FALSE",
                     I_Spare14 := "FALSE",
                     H_IAnim => #"H_GBLiftTable2Pos1S3Det-C".H_DetSetIAnim[1].H_DWord);
   END_IF;
END_REGION

REGION Network 29: **** 4.6 - Machine status - Indication **** LSpdDetSetIAnim / **** 4.6 - Machine status - Indication **** DetSetCheck IAnim
   // Icon animation
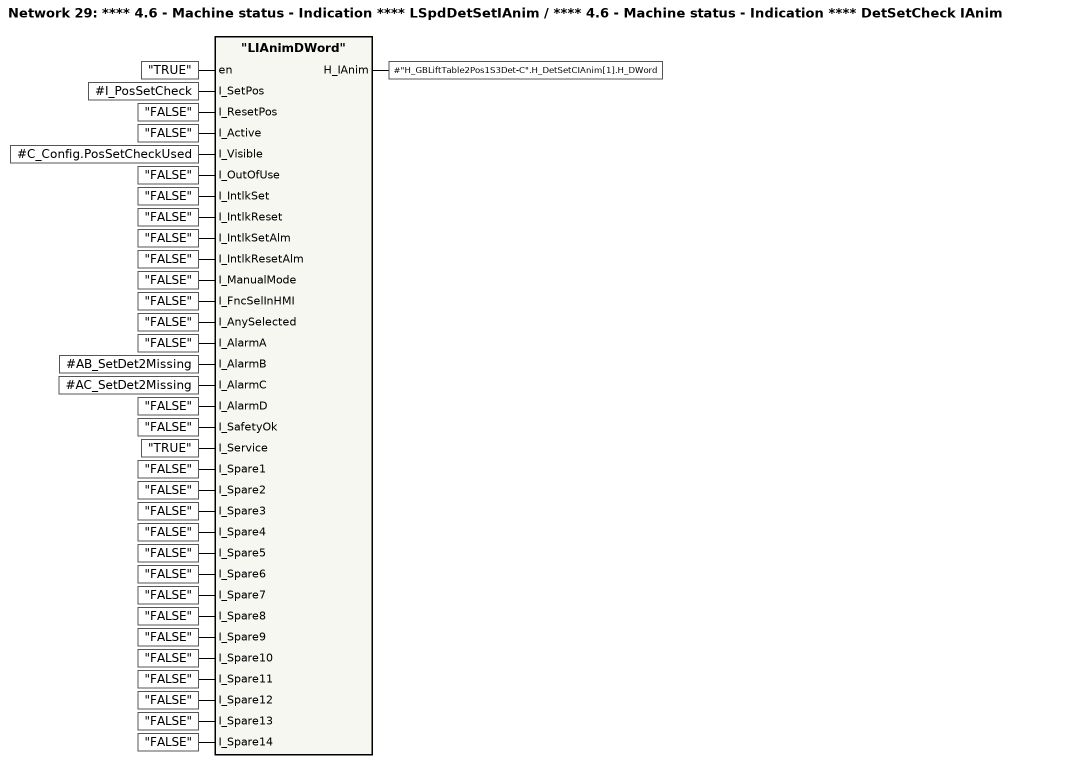
   IF "TRUE" THEN
       "LIAnimDWord"(I_SetPos := #I_PosSetCheck,
                     I_ResetPos := "FALSE",
                     I_Active := "FALSE",
                     I_Visible := #C_Config.PosSetCheckUsed,
                     I_OutOfUse := "FALSE",
                     I_IntlkSet := "FALSE",
                     I_IntlkReset := "FALSE",
                     I_IntlkSetAlm := "FALSE",
                     I_IntlkResetAlm := "FALSE",
                     I_ManualMode := "FALSE",
                     I_FncSelInHMI := "FALSE",
                     I_AnySelected := "FALSE",
                     I_AlarmA := "FALSE",
                     I_AlarmB := #AB_SetDet2Missing,
                     I_AlarmC := #AC_SetDet2Missing,
                     I_AlarmD := "FALSE",
                     I_SafetyOk := "FALSE",
                     I_Service := "TRUE",
                     I_Spare1 := "FALSE",
                     I_Spare2 := "FALSE",
                     I_Spare3 := "FALSE",
                     I_Spare4 := "FALSE",
                     I_Spare5 := "FALSE",
                     I_Spare6 := "FALSE",
                     I_Spare7 := "FALSE",
                     I_Spare8 := "FALSE",
                     I_Spare9 := "FALSE",
                     I_Spare10 := "FALSE",
                     I_Spare11 := "FALSE",
                     I_Spare12 := "FALSE",
                     I_Spare13 := "FALSE",
                     I_Spare14 := "FALSE",
                     H_IAnim => #"H_GBLiftTable2Pos1S3Det-C".H_DetSetCIAnim[1].H_DWord);
   END_IF;
END_REGION

REGION Network 30: **** 4.6 - Machine status - Indication **** ResetDet1IAnim / **** 4.6 - Machine status - Indication **** ResetDetIAnim / **** 4.6 - Machine status - Indication **** DetRes IAnim
   // Icon animation
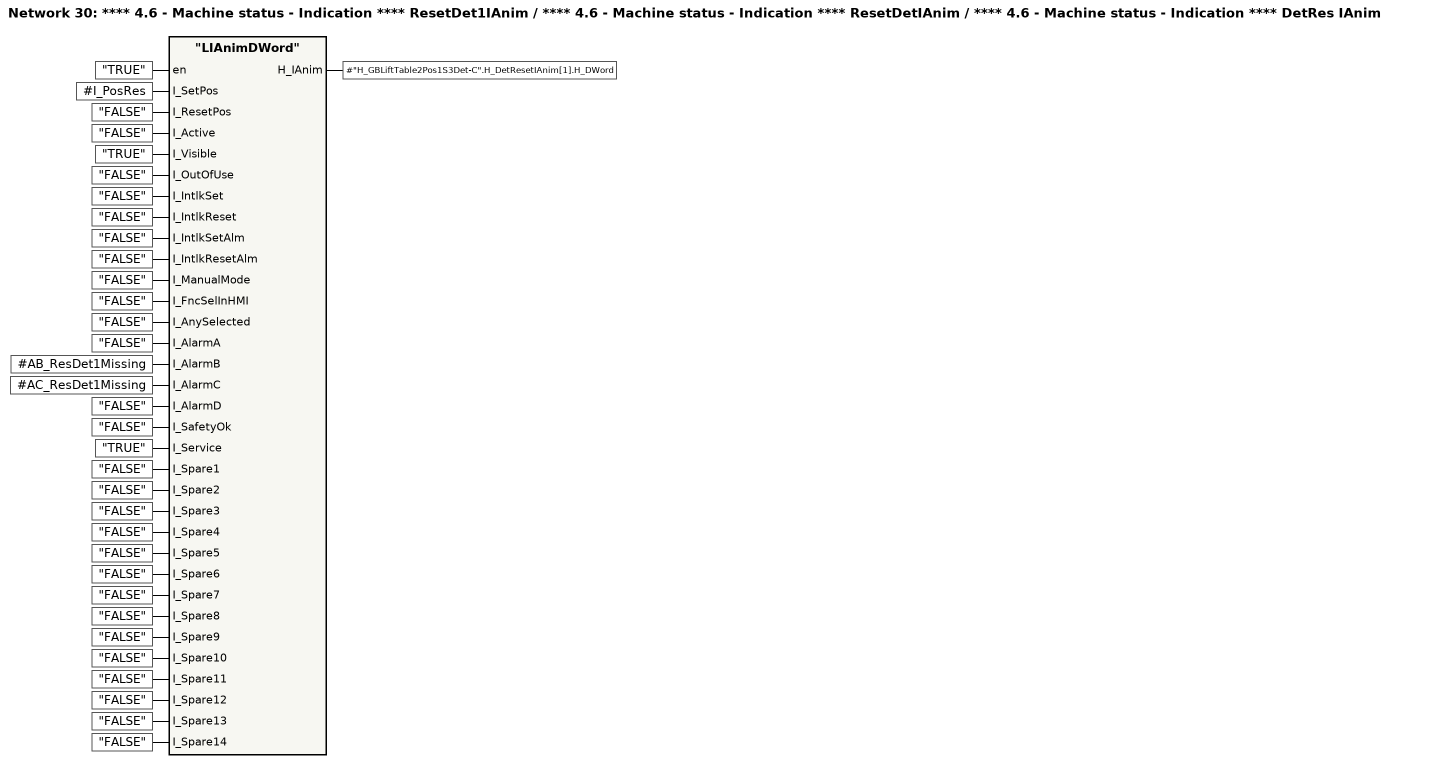
   IF "TRUE" THEN
       "LIAnimDWord"(I_SetPos := #I_PosRes,
                     I_ResetPos := "FALSE",
                     I_Active := "FALSE",
                     I_Visible := "TRUE",
                     I_OutOfUse := "FALSE",
                     I_IntlkSet := "FALSE",
                     I_IntlkReset := "FALSE",
                     I_IntlkSetAlm := "FALSE",
                     I_IntlkResetAlm := "FALSE",
                     I_ManualMode := "FALSE",
                     I_FncSelInHMI := "FALSE",
                     I_AnySelected := "FALSE",
                     I_AlarmA := "FALSE",
                     I_AlarmB := #AB_ResDet1Missing,
                     I_AlarmC := #AC_ResDet1Missing,
                     I_AlarmD := "FALSE",
                     I_SafetyOk := "FALSE",
                     I_Service := "TRUE",
                     I_Spare1 := "FALSE",
                     I_Spare2 := "FALSE",
                     I_Spare3 := "FALSE",
                     I_Spare4 := "FALSE",
                     I_Spare5 := "FALSE",
                     I_Spare6 := "FALSE",
                     I_Spare7 := "FALSE",
                     I_Spare8 := "FALSE",
                     I_Spare9 := "FALSE",
                     I_Spare10 := "FALSE",
                     I_Spare11 := "FALSE",
                     I_Spare12 := "FALSE",
                     I_Spare13 := "FALSE",
                     I_Spare14 := "FALSE",
                     H_IAnim => #"H_GBLiftTable2Pos1S3Det-C".H_DetResetIAnim[1].H_DWord);
   END_IF;
END_REGION

REGION Network 31: **** 4.6 - Machine status - Indication **** LSpdDetResIAnim / **** 4.6 - Machine status - Indication **** DetResCheck IAnim
   // Icon animation
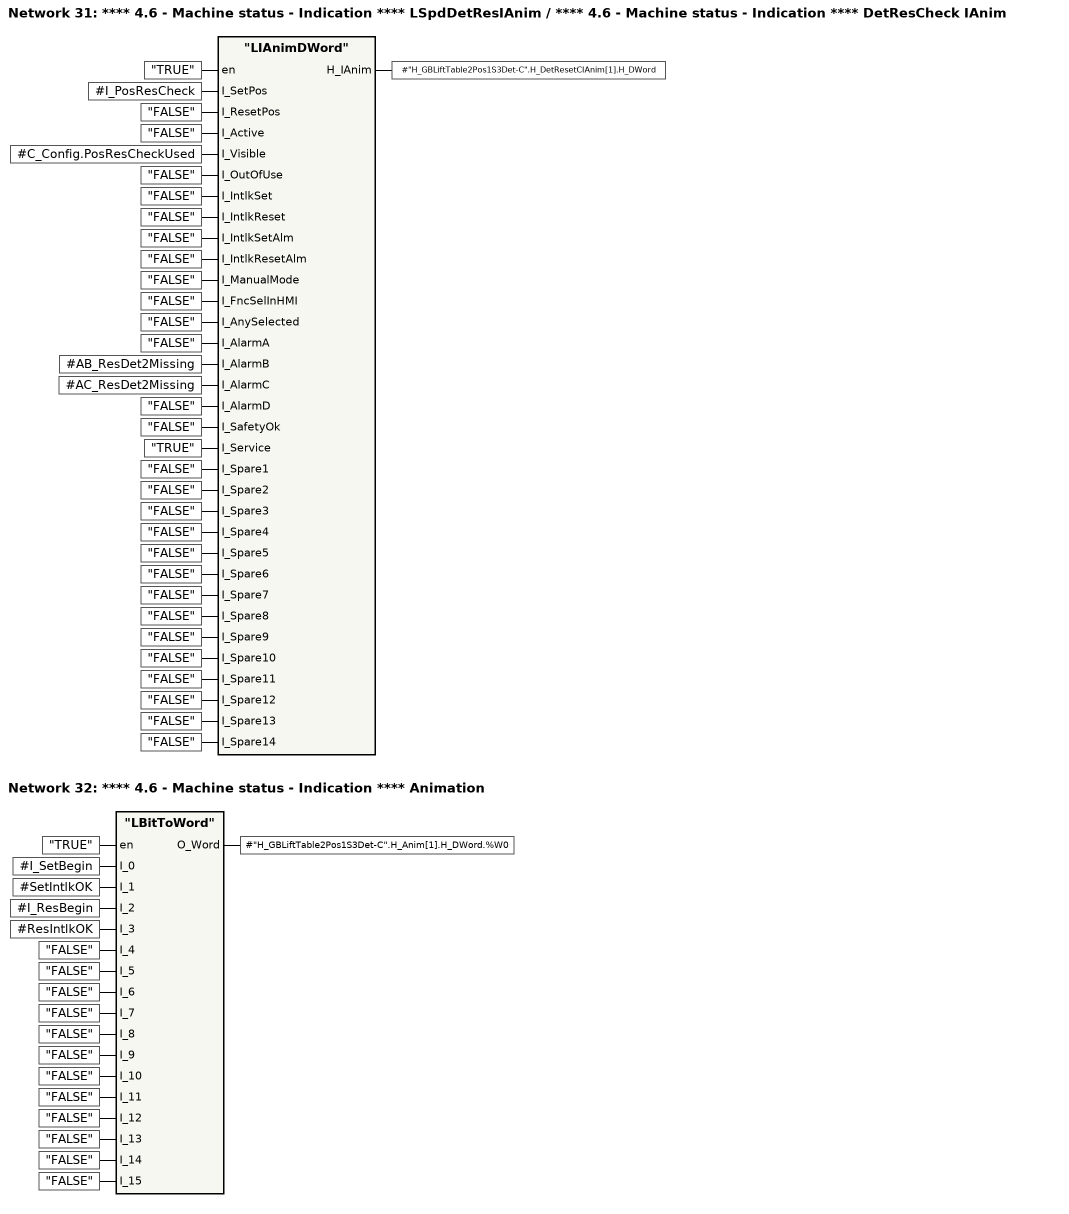
   IF "TRUE" THEN
       "LIAnimDWord"(I_SetPos := #I_PosResCheck,
                     I_ResetPos := "FALSE",
                     I_Active := "FALSE",
                     I_Visible := #C_Config.PosResCheckUsed,
                     I_OutOfUse := "FALSE",
                     I_IntlkSet := "FALSE",
                     I_IntlkReset := "FALSE",
                     I_IntlkSetAlm := "FALSE",
                     I_IntlkResetAlm := "FALSE",
                     I_ManualMode := "FALSE",
                     I_FncSelInHMI := "FALSE",
                     I_AnySelected := "FALSE",
                     I_AlarmA := "FALSE",
                     I_AlarmB := #AB_ResDet2Missing,
                     I_AlarmC := #AC_ResDet2Missing,
                     I_AlarmD := "FALSE",
                     I_SafetyOk := "FALSE",
                     I_Service := "TRUE",
                     I_Spare1 := "FALSE",
                     I_Spare2 := "FALSE",
                     I_Spare3 := "FALSE",
                     I_Spare4 := "FALSE",
                     I_Spare5 := "FALSE",
                     I_Spare6 := "FALSE",
                     I_Spare7 := "FALSE",
                     I_Spare8 := "FALSE",
                     I_Spare9 := "FALSE",
                     I_Spare10 := "FALSE",
                     I_Spare11 := "FALSE",
                     I_Spare12 := "FALSE",
                     I_Spare13 := "FALSE",
                     I_Spare14 := "FALSE",
                     H_IAnim => #"H_GBLiftTable2Pos1S3Det-C".H_DetResetCIAnim[1].H_DWord);
   END_IF;
END_REGION

REGION Network 32: **** 4.6 - Machine status - Indication **** Animation
   // Animation
   IF "TRUE" THEN
       "LBitToWord"(I_0 := #I_SetBegin,
                    I_1 := #SetIntlkOK,
                    I_2 := #I_ResBegin,
                    I_3 := #ResIntlkOK,
                    I_4 := "FALSE",
                    I_5 := "FALSE",
                    I_6 := "FALSE",
                    I_7 := "FALSE",
                    I_8 := "FALSE",
                    I_9 := "FALSE",
                    I_10 := "FALSE",
                    I_11 := "FALSE",
                    I_12 := "FALSE",
                    I_13 := "FALSE",
                    I_14 := "FALSE",
                    I_15 := "FALSE",
                    O_Word => #"H_GBLiftTable2Pos1S3Det-C".H_Anim[1].H_DWord.%W0);
   END_IF;
END_REGION

REGION Network 33: **** 4.6 - Machine status - Indication **** Animation
   // Animation
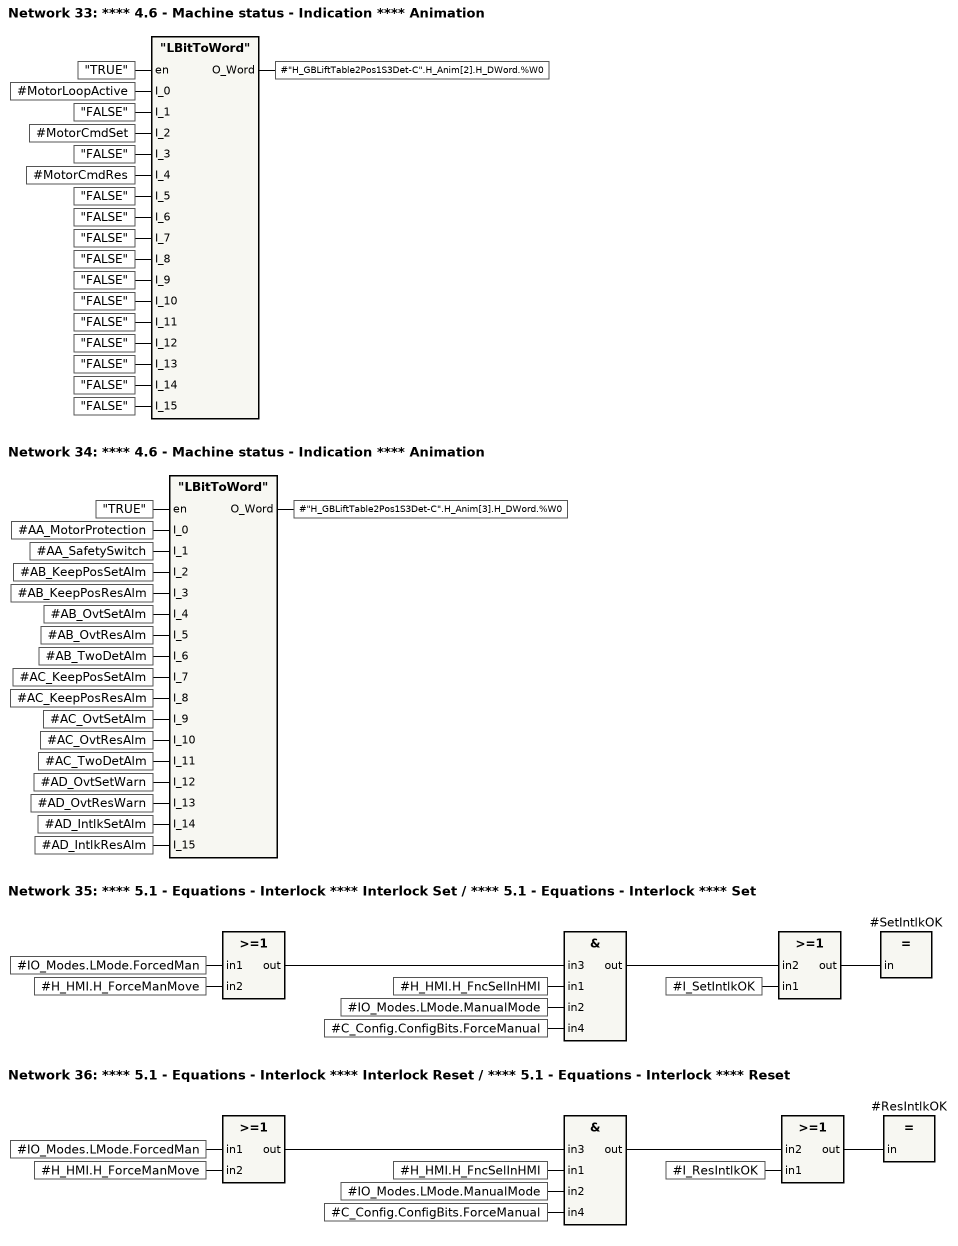
   IF "TRUE" THEN
       "LBitToWord"(I_0 := #MotorLoopActive,
                    I_1 := "FALSE",
                    I_2 := #MotorCmdSet,
                    I_3 := "FALSE",
                    I_4 := #MotorCmdRes,
                    I_5 := "FALSE",
                    I_6 := "FALSE",
                    I_7 := "FALSE",
                    I_8 := "FALSE",
                    I_9 := "FALSE",
                    I_10 := "FALSE",
                    I_11 := "FALSE",
                    I_12 := "FALSE",
                    I_13 := "FALSE",
                    I_14 := "FALSE",
                    I_15 := "FALSE",
                    O_Word => #"H_GBLiftTable2Pos1S3Det-C".H_Anim[2].H_DWord.%W0);
   END_IF;
END_REGION

REGION Network 34: **** 4.6 - Machine status - Indication **** Animation
   // Animation
   IF "TRUE" THEN
       "LBitToWord"(I_0 := #AA_MotorProtection,
                    I_1 := #AA_SafetySwitch,
                    I_2 := #AB_KeepPosSetAlm,
                    I_3 := #AB_KeepPosResAlm,
                    I_4 := #AB_OvtSetAlm,
                    I_5 := #AB_OvtResAlm,
                    I_6 := #AB_TwoDetAlm,
                    I_7 := #AC_KeepPosSetAlm,
                    I_8 := #AC_KeepPosResAlm,
                    I_9 := #AC_OvtSetAlm,
                    I_10 := #AC_OvtResAlm,
                    I_11 := #AC_TwoDetAlm,
                    I_12 := #AD_OvtSetWarn,
                    I_13 := #AD_OvtResWarn,
                    I_14 := #AD_IntlkSetAlm,
                    I_15 := #AD_IntlkResAlm,
                    O_Word => #"H_GBLiftTable2Pos1S3Det-C".H_Anim[3].H_DWord.%W0);
   END_IF;
END_REGION

REGION Network 35: **** 5.1 - Equations - Interlock **** Interlock Set / **** 5.1 - Equations - Interlock **** Set
   // Interlock
   #SetIntlkOK := ((#IO_Modes.LMode.ForcedMan OR #H_HMI.H_ForceManMove) AND #H_HMI.H_FncSelInHMI AND #IO_Modes.LMode.ManualMode AND #C_Config.ConfigBits.ForceManual) OR #I_SetIntlkOK;
END_REGION

REGION Network 36: **** 5.1 - Equations - Interlock **** Interlock Reset / **** 5.1 - Equations - Interlock **** Reset
   // Interlock
   #ResIntlkOK := ((#IO_Modes.LMode.ForcedMan OR #H_HMI.H_ForceManMove) AND #H_HMI.H_FncSelInHMI AND #IO_Modes.LMode.ManualMode AND #C_Config.ConfigBits.ForceManual) OR #I_ResIntlkOK;
END_REGION

REGION Network 37: **** 7.3 - Submodule - Machine **** LMovFunc2Pos
   // LMovFunc2Pos2s / LMovFunc2Pos
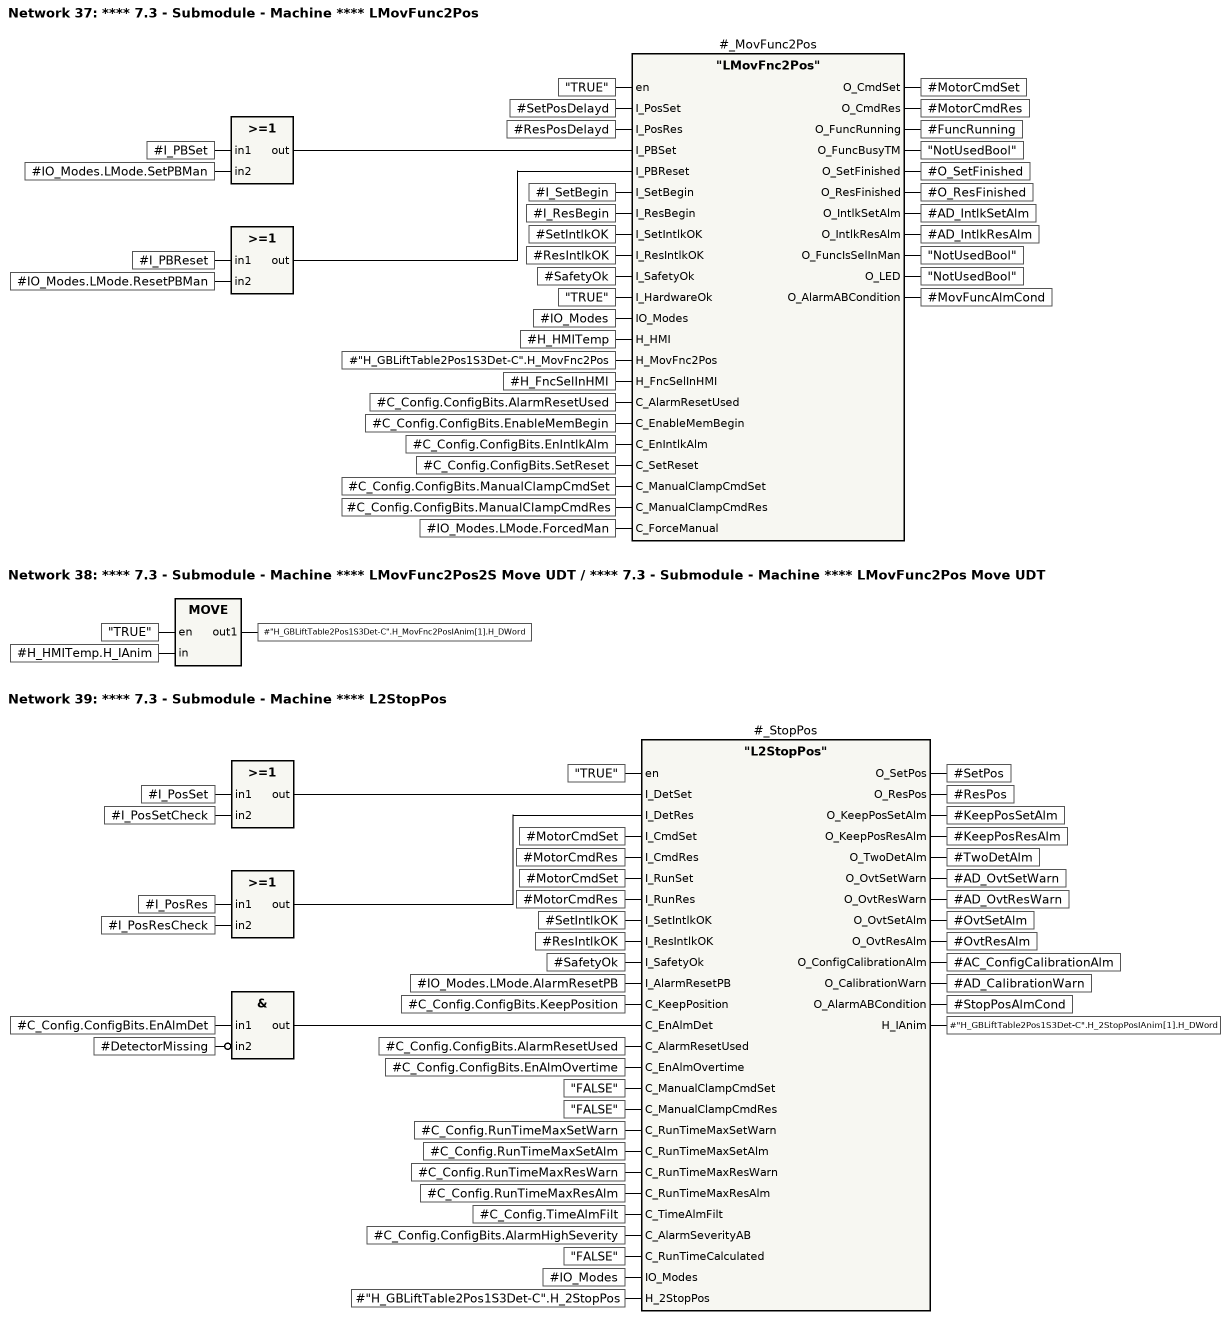
   IF "TRUE" THEN
       #_MovFunc2Pos(I_PosSet := #SetPosDelayd,   // "LMovFnc2Pos"
                     I_PosRes := #ResPosDelayd,
                     I_PBSet := #I_PBSet OR #IO_Modes.LMode.SetPBMan,
                     I_PBReset := #I_PBReset OR #IO_Modes.LMode.ResetPBMan,
                     I_SetBegin := #I_SetBegin,
                     I_ResBegin := #I_ResBegin,
                     I_SetIntlkOK := #SetIntlkOK,
                     I_ResIntlkOK := #ResIntlkOK,
                     I_SafetyOk := #SafetyOk,
                     I_HardwareOk := "TRUE",
                     IO_Modes := #IO_Modes,
                     H_HMI := #H_HMITemp,
                     H_MovFnc2Pos := #"H_GBLiftTable2Pos1S3Det-C".H_MovFnc2Pos,
                     H_FncSelInHMI := #H_FncSelInHMI,
                     C_AlarmResetUsed := #C_Config.ConfigBits.AlarmResetUsed,
                     C_EnableMemBegin := #C_Config.ConfigBits.EnableMemBegin,
                     C_EnIntlkAlm := #C_Config.ConfigBits.EnIntlkAlm,
                     C_SetReset := #C_Config.ConfigBits.SetReset,
                     C_ManualClampCmdSet := #C_Config.ConfigBits.ManualClampCmdSet,
                     C_ManualClampCmdRes := #C_Config.ConfigBits.ManualClampCmdRes,
                     C_ForceManual := #IO_Modes.LMode.ForcedMan,
                     O_CmdSet => #MotorCmdSet,
                     O_CmdRes => #MotorCmdRes,
                     O_FuncRunning => #FuncRunning,
                     O_FuncBusyTM => "NotUsedBool",
                     O_SetFinished => #O_SetFinished,
                     O_ResFinished => #O_ResFinished,
                     O_IntlkSetAlm => #AD_IntlkSetAlm,
                     O_IntlkResAlm => #AD_IntlkResAlm,
                     O_FuncIsSelInMan => "NotUsedBool",
                     O_LED => "NotUsedBool",
                     O_AlarmABCondition => #MovFuncAlmCond);
   END_IF;
END_REGION

REGION Network 38: **** 7.3 - Submodule - Machine **** LMovFunc2Pos2S Move UDT / **** 7.3 - Submodule - Machine **** LMovFunc2Pos Move UDT
   // LMovFunc2Pos2S Move UDT
   IF "TRUE" THEN #"H_GBLiftTable2Pos1S3Det-C".H_MovFnc2PosIAnim[1].H_DWord := #H_HMITemp.H_IAnim; END_IF;
END_REGION

REGION Network 39: **** 7.3 - Submodule - Machine **** L2StopPos
   // L2StopPos
   IF "TRUE" THEN
       #_StopPos(I_DetSet := #I_PosSet OR #I_PosSetCheck,   // "L2StopPos"
                 I_DetRes := #I_PosRes OR #I_PosResCheck,
                 I_CmdSet := #MotorCmdSet,
                 I_CmdRes := #MotorCmdRes,
                 I_RunSet := #MotorCmdSet,
                 I_RunRes := #MotorCmdRes,
                 I_SetIntlkOK := #SetIntlkOK,
                 I_ResIntlkOK := #ResIntlkOK,
                 I_SafetyOk := #SafetyOk,
                 I_AlarmResetPB := #IO_Modes.LMode.AlarmResetPB,
                 C_KeepPosition := #C_Config.ConfigBits.KeepPosition,
                 C_EnAlmDet := #C_Config.ConfigBits.EnAlmDet AND NOT #DetectorMissing,
                 C_AlarmResetUsed := #C_Config.ConfigBits.AlarmResetUsed,
                 C_EnAlmOvertime := #C_Config.ConfigBits.EnAlmOvertime,
                 C_ManualClampCmdSet := "FALSE",
                 C_ManualClampCmdRes := "FALSE",
                 C_RunTimeMaxSetWarn := #C_Config.RunTimeMaxSetWarn,
                 C_RunTimeMaxSetAlm := #C_Config.RunTimeMaxSetAlm,
                 C_RunTimeMaxResWarn := #C_Config.RunTimeMaxResWarn,
                 C_RunTimeMaxResAlm := #C_Config.RunTimeMaxResAlm,
                 C_TimeAlmFilt := #C_Config.TimeAlmFilt,
                 C_AlarmSeverityAB := #C_Config.ConfigBits.AlarmHighSeverity,
                 C_RunTimeCalculated := "FALSE",
                 IO_Modes := #IO_Modes,
                 H_2StopPos := #"H_GBLiftTable2Pos1S3Det-C".H_2StopPos,
                 O_SetPos => #SetPos,
                 O_ResPos => #ResPos,
                 O_KeepPosSetAlm => #KeepPosSetAlm,
                 O_KeepPosResAlm => #KeepPosResAlm,
                 O_TwoDetAlm => #TwoDetAlm,
                 O_OvtSetWarn => #AD_OvtSetWarn,
                 O_OvtResWarn => #AD_OvtResWarn,
                 O_OvtSetAlm => #OvtSetAlm,
                 O_OvtResAlm => #OvtResAlm,
                 O_ConfigCalibrationAlm => #AC_ConfigCalibrationAlm,
                 O_CalibrationWarn => #AD_CalibrationWarn,
                 O_AlarmABCondition => #StopPosAlmCond,
                 H_IAnim => #"H_GBLiftTable2Pos1S3Det-C".H_2StopPosIAnim[1].H_DWord);
   END_IF;
END_REGION

REGION Network 40: **** 7.3 - Submodule - Machine **** Motor Loop MOVIFIT-FC / **** 7.3 - Submodule - Machine **** Motor Loop
   // Motor loop G120
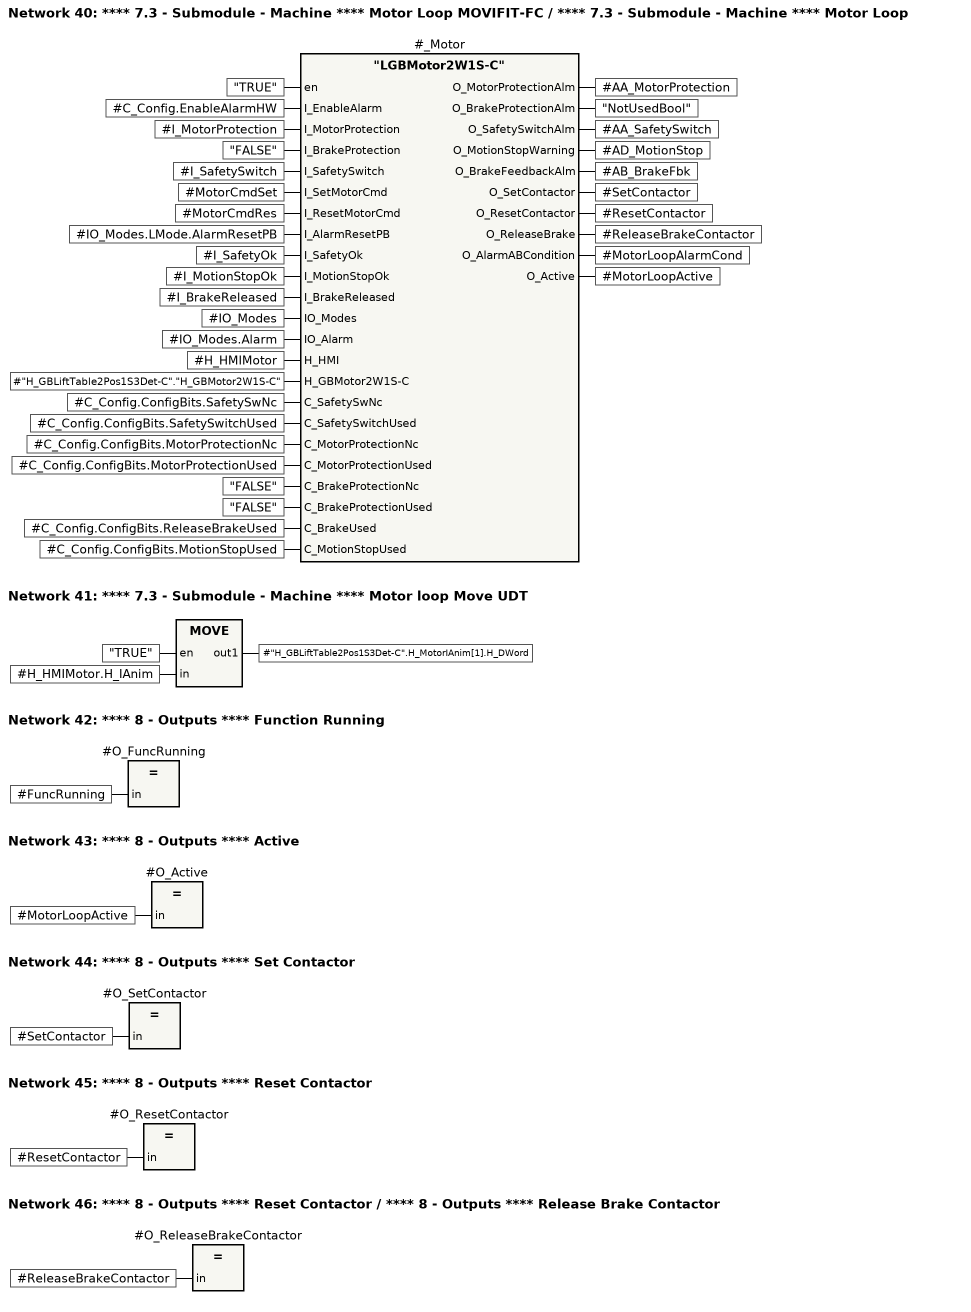
   IF "TRUE" THEN
       #_Motor(I_EnableAlarm := #C_Config.EnableAlarmHW,   // "LGBMotor2W1S-C"
               I_MotorProtection := #I_MotorProtection,
               I_BrakeProtection := "FALSE",
               I_SafetySwitch := #I_SafetySwitch,
               I_SetMotorCmd := #MotorCmdSet,
               I_ResetMotorCmd := #MotorCmdRes,
               I_AlarmResetPB := #IO_Modes.LMode.AlarmResetPB,
               I_SafetyOk := #I_SafetyOk,
               I_MotionStopOk := #I_MotionStopOk,
               I_BrakeReleased := #I_BrakeReleased,
               IO_Modes := #IO_Modes,
               IO_Alarm := #IO_Modes.Alarm,
               H_HMI := #H_HMIMotor,
               "H_GBMotor2W1S-C" := #"H_GBLiftTable2Pos1S3Det-C"."H_GBMotor2W1S-C",
               C_SafetySwNc := #C_Config.ConfigBits.SafetySwNc,
               C_SafetySwitchUsed := #C_Config.ConfigBits.SafetySwitchUsed,
               C_MotorProtectionNc := #C_Config.ConfigBits.MotorProtectionNc,
               C_MotorProtectionUsed := #C_Config.ConfigBits.MotorProtectionUsed,
               C_BrakeProtectionNc := "FALSE",
               C_BrakeProtectionUsed := "FALSE",
               C_BrakeUsed := #C_Config.ConfigBits.ReleaseBrakeUsed,
               C_MotionStopUsed := #C_Config.ConfigBits.MotionStopUsed,
               O_MotorProtectionAlm => #AA_MotorProtection,
               O_BrakeProtectionAlm => "NotUsedBool",
               O_SafetySwitchAlm => #AA_SafetySwitch,
               O_MotionStopWarning => #AD_MotionStop,
               O_BrakeFeedbackAlm => #AB_BrakeFbk,
               O_SetContactor => #SetContactor,
               O_ResetContactor => #ResetContactor,
               O_ReleaseBrake => #ReleaseBrakeContactor,
               O_AlarmABCondition => #MotorLoopAlarmCond,
               O_Active => #MotorLoopActive);
   END_IF;
END_REGION

REGION Network 41: **** 7.3 - Submodule - Machine **** Motor loop Move UDT
   IF "TRUE" THEN #"H_GBLiftTable2Pos1S3Det-C".H_MotorIAnim[1].H_DWord := #H_HMIMotor.H_IAnim; END_IF;
END_REGION

REGION Network 42: **** 8 - Outputs **** Function Running
   // Function Running
   #O_FuncRunning := #FuncRunning;
END_REGION

REGION Network 43: **** 8 - Outputs **** Active
   // Motor Loop active
   #O_Active := #MotorLoopActive;
END_REGION

REGION Network 44: **** 8 - Outputs **** Set Contactor
   // Set Contactor
   #O_SetContactor := #SetContactor;
END_REGION

REGION Network 45: **** 8 - Outputs **** Reset Contactor
   // Reset Contactor
   #O_ResetContactor := #ResetContactor;
END_REGION

REGION Network 46: **** 8 - Outputs **** Reset Contactor / **** 8 - Outputs **** Release Brake Contactor
   // Reset Contactor / Release Brake Contactor
   #O_ReleaseBrakeContactor := #ReleaseBrakeContactor;
END_REGION

REGION Network 47: **** 8 - Outputs **** Summary Position Set
   // Summary Position Set
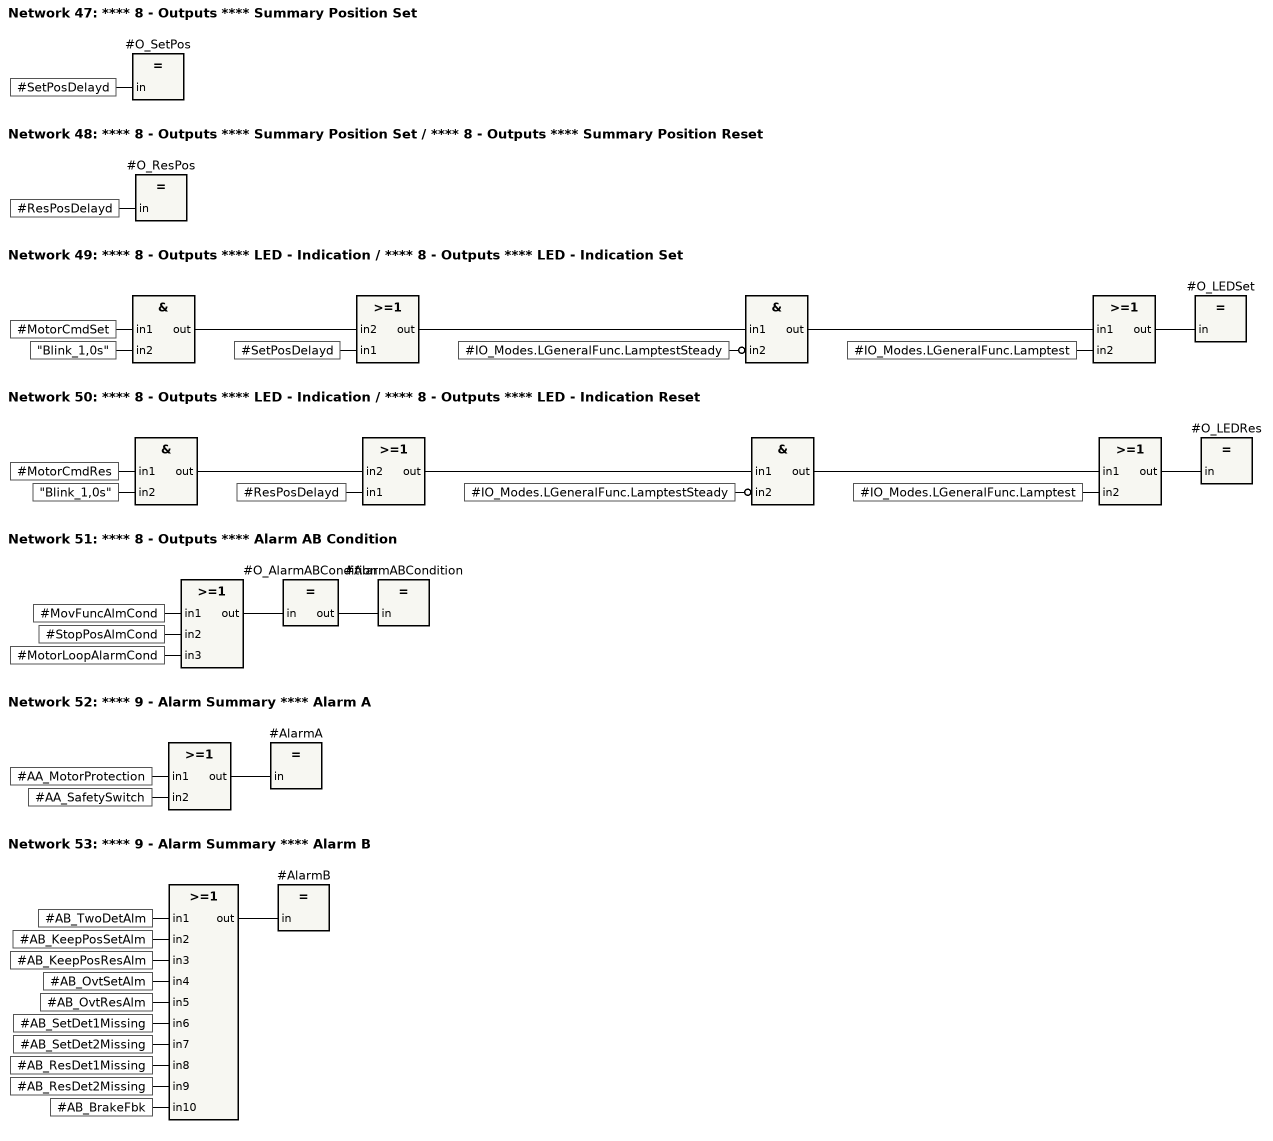
   #O_SetPos := #SetPosDelayd;
END_REGION

REGION Network 48: **** 8 - Outputs **** Summary Position Set / **** 8 - Outputs **** Summary Position Reset
   // Summary Position Reset
   #O_ResPos := #ResPosDelayd;
END_REGION

REGION Network 49: **** 8 - Outputs **** LED - Indication / **** 8 - Outputs **** LED - Indication Set
   // LED - Indication
   #O_LEDSet := (((#MotorCmdSet AND "Blink_1,0s") OR #SetPosDelayd) AND NOT #IO_Modes.LGeneralFunc.LamptestSteady) OR #IO_Modes.LGeneralFunc.Lamptest;
END_REGION

REGION Network 50: **** 8 - Outputs **** LED - Indication / **** 8 - Outputs **** LED - Indication Reset
   // LED - Indication
   #O_LEDRes := (((#MotorCmdRes AND "Blink_1,0s") OR #ResPosDelayd) AND NOT #IO_Modes.LGeneralFunc.LamptestSteady) OR #IO_Modes.LGeneralFunc.Lamptest;
END_REGION

REGION Network 51: **** 8 - Outputs **** Alarm AB Condition
   // Alarm AB condition
   #O_AlarmABCondition := #MovFuncAlmCond OR #StopPosAlmCond OR #MotorLoopAlarmCond;
   #AlarmABCondition := #O_AlarmABCondition;
END_REGION

REGION Network 52: **** 9 - Alarm Summary **** Alarm A
   // Alarms A
   #AlarmA := #AA_MotorProtection OR #AA_SafetySwitch;
END_REGION

REGION Network 53: **** 9 - Alarm Summary **** Alarm B
   // Alarms B
   #AlarmB := #AB_TwoDetAlm OR #AB_KeepPosSetAlm OR #AB_KeepPosResAlm OR #AB_OvtSetAlm OR #AB_OvtResAlm OR #AB_SetDet1Missing OR #AB_SetDet2Missing OR #AB_ResDet1Missing OR #AB_ResDet2Missing OR #AB_BrakeFbk;
END_REGION

REGION Network 54: **** 9 - Alarm Summary **** Alarm C
   // Alarms C
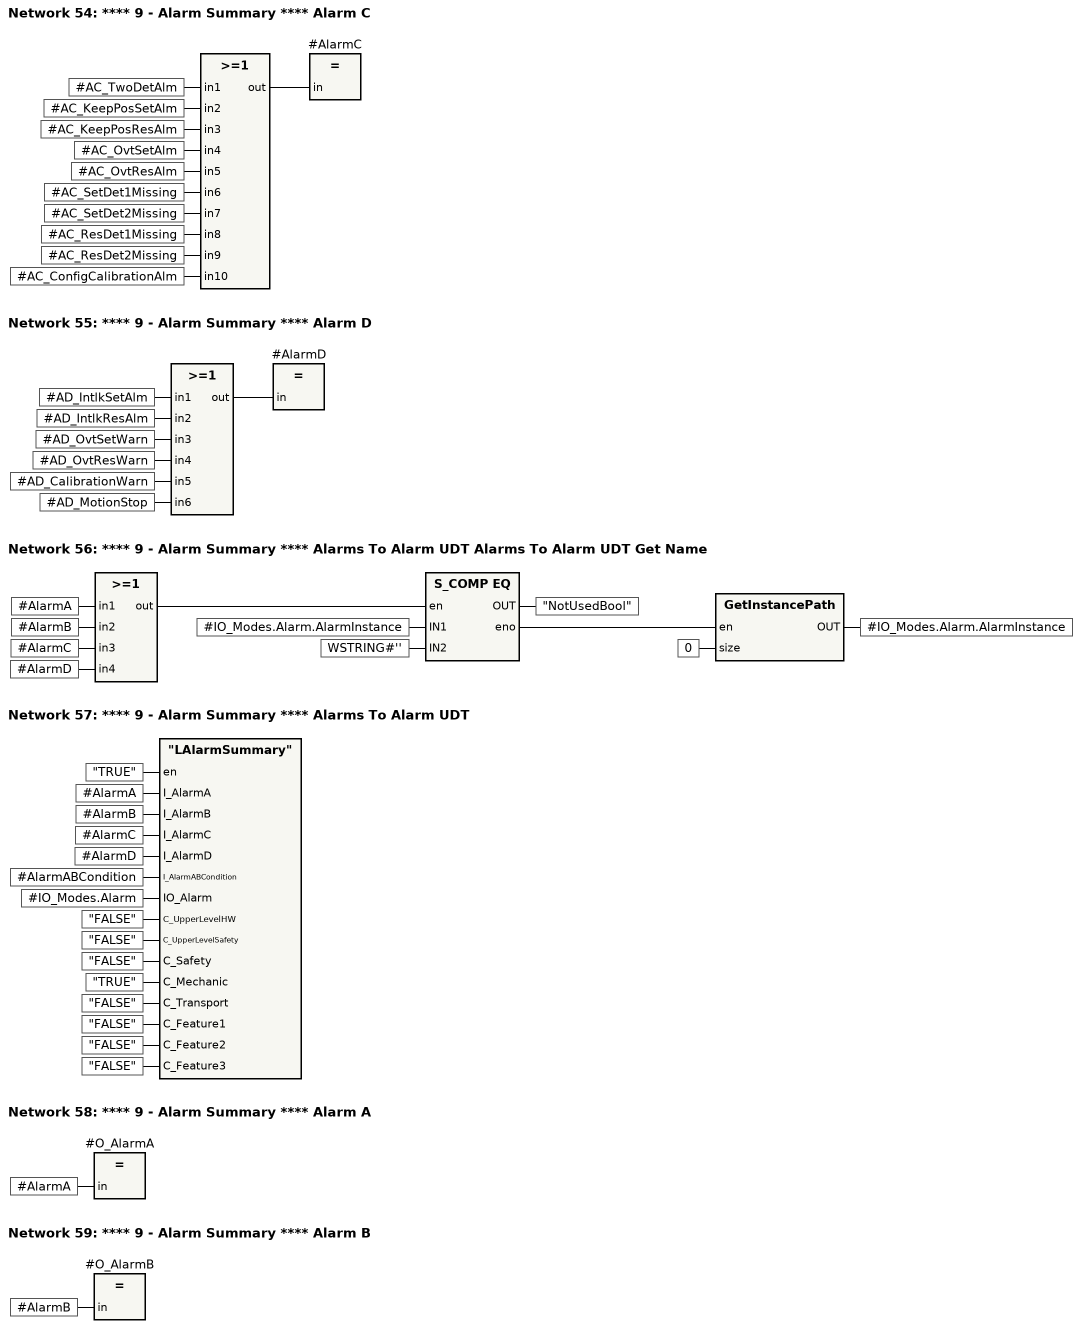
   #AlarmC := #AC_TwoDetAlm OR #AC_KeepPosSetAlm OR #AC_KeepPosResAlm OR #AC_OvtSetAlm OR #AC_OvtResAlm OR #AC_SetDet1Missing OR #AC_SetDet2Missing OR #AC_ResDet1Missing OR #AC_ResDet2Missing OR #AC_ConfigCalibrationAlm;
END_REGION

REGION Network 55: **** 9 - Alarm Summary **** Alarm D
   // Alarms D
   #AlarmD := #AD_IntlkSetAlm OR #AD_IntlkResAlm OR #AD_OvtSetWarn OR #AD_OvtResWarn OR #AD_CalibrationWarn OR #AD_MotionStop;
END_REGION

REGION Network 56: **** 9 - Alarm Summary **** Alarms To Alarm UDT Alarms To Alarm UDT Get Name
   // Alarm D
   S_COMP(EN := #AlarmA OR #AlarmB OR #AlarmC OR #AlarmD,
          IN1 := #IO_Modes.Alarm.AlarmInstance,
          IN2 := WSTRING#'',
          OUT => "NotUsedBool",
          ENO => #_w1);
   IF #_w1 THEN GetInstancePath(size := 0, OUT => #IO_Modes.Alarm.AlarmInstance); END_IF;
END_REGION

REGION Network 57: **** 9 - Alarm Summary **** Alarms To Alarm UDT
   // Alarm D
   IF "TRUE" THEN
       "LAlarmSummary"(I_AlarmA := #AlarmA,
                       I_AlarmB := #AlarmB,
                       I_AlarmC := #AlarmC,
                       I_AlarmD := #AlarmD,
                       I_AlarmABCondition := #AlarmABCondition,
                       IO_Alarm := #IO_Modes.Alarm,
                       C_UpperLevelHW := "FALSE",
                       C_UpperLevelSafety := "FALSE",
                       C_Safety := "FALSE",
                       C_Mechanic := "TRUE",
                       C_Transport := "FALSE",
                       C_Feature1 := "FALSE",
                       C_Feature2 := "FALSE",
                       C_Feature3 := "FALSE");
   END_IF;
END_REGION

REGION Network 58: **** 9 - Alarm Summary **** Alarm A
   // Alarm A
   #O_AlarmA := #AlarmA;
END_REGION

REGION Network 59: **** 9 - Alarm Summary **** Alarm B
   // Alarm B
   #O_AlarmB := #AlarmB;
END_REGION

REGION Network 60: **** 9 - Alarm Summary **** Alarm C
   // Alarm C
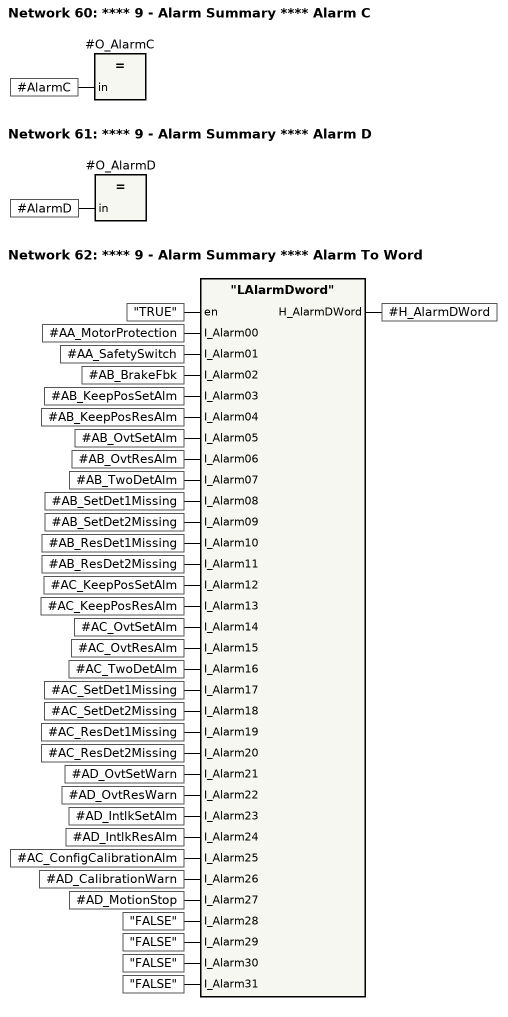
   #O_AlarmC := #AlarmC;
END_REGION

REGION Network 61: **** 9 - Alarm Summary **** Alarm D
   // Alarm D
   #O_AlarmD := #AlarmD;
END_REGION

REGION Network 62: **** 9 - Alarm Summary **** Alarm To Word
   // Alarm To Word
   IF "TRUE" THEN
       "LAlarmDword"(I_Alarm00 := #AA_MotorProtection,
                     I_Alarm01 := #AA_SafetySwitch,
                     I_Alarm02 := #AB_BrakeFbk,
                     I_Alarm03 := #AB_KeepPosSetAlm,
                     I_Alarm04 := #AB_KeepPosResAlm,
                     I_Alarm05 := #AB_OvtSetAlm,
                     I_Alarm06 := #AB_OvtResAlm,
                     I_Alarm07 := #AB_TwoDetAlm,
                     I_Alarm08 := #AB_SetDet1Missing,
                     I_Alarm09 := #AB_SetDet2Missing,
                     I_Alarm10 := #AB_ResDet1Missing,
                     I_Alarm11 := #AB_ResDet2Missing,
                     I_Alarm12 := #AC_KeepPosSetAlm,
                     I_Alarm13 := #AC_KeepPosResAlm,
                     I_Alarm14 := #AC_OvtSetAlm,
                     I_Alarm15 := #AC_OvtResAlm,
                     I_Alarm16 := #AC_TwoDetAlm,
                     I_Alarm17 := #AC_SetDet1Missing,
                     I_Alarm18 := #AC_SetDet2Missing,
                     I_Alarm19 := #AC_ResDet1Missing,
                     I_Alarm20 := #AC_ResDet2Missing,
                     I_Alarm21 := #AD_OvtSetWarn,
                     I_Alarm22 := #AD_OvtResWarn,
                     I_Alarm23 := #AD_IntlkSetAlm,
                     I_Alarm24 := #AD_IntlkResAlm,
                     I_Alarm25 := #AC_ConfigCalibrationAlm,
                     I_Alarm26 := #AD_CalibrationWarn,
                     I_Alarm27 := #AD_MotionStop,
                     I_Alarm28 := "FALSE",
                     I_Alarm29 := "FALSE",
                     I_Alarm30 := "FALSE",
                     I_Alarm31 := "FALSE",
                     H_AlarmDWord => #H_AlarmDWord);
   END_IF;
END_REGION
END_FUNCTION_BLOCK
